// ---- PLC_MOTION/FLYING_SAW/class/FB_FlyingCtrl.TcPOU
FUNCTION_BLOCK FB_FlyingCtrl EXTENDS FB_FlyingBase IMPLEMENTS I_Fly_Ctrl
VAR
  _eInit                    : E_PROGRESS;
  _nAxisIndex               : UINT;       // know thyself
  _nMasterIndex             : UINT;       // to whom must I answer?

  // get interface from McAxis for access to Reset, Enable, Disable, Halt
  _ItfMcAxis                : ARRAY[1..PLC_CONSTANT.MAX_AXIS] OF I_McAxis;

  // pointers to all; access required for coupling; access by index
  _Ctrl                     : POINTER TO ARRAY[1..PLC_CONSTANT.MAX_AXIS] OF ST_FLY_CTRL;    // contains command to be executed
  _State                    : POINTER TO ARRAY[1..PLC_CONSTANT.MAX_AXIS] OF ST_FLY_STATE;   // mirrors command with added result

  //_Info                     : POINTER TO ARRAY[1..PLC_CONSTANT.MAX_AXIS] OF ST_FLY_INFO;    // Read Info Data
  _Data                     : POINTER TO ARRAY[1..PLC_CONSTANT.MAX_AXIS] OF ST_FLY_DATA;    // fLYINGsAW parameters

  _MoveData                 : POINTER TO ARRAY[1..PLC_CONSTANT.MAX_AXIS] OF ST_AXIS_MOVE_DATA;   // dynamic parameters

  _Options                  : POINTER TO ARRAY[1..PLC_CONSTANT.MAX_AXIS] OF ST_FLY_OPTIONS; // gear in slave options

  // local copies of command
  _eCmd,
  _eCmdOld                  : E_AXIS_CTRL;

  // execution state
  _eResult                  : E_PROGRESS;   // result of execution state
  _eResultOld               : E_PROGRESS;   // old result for detecting change
  _eState                   : E_AXIS_STATE; // execution state
END_VAR

PROPERTY AxisCtrl : pointer to ARRAY[1..PLC_CONSTANT.MAX_AXIS] OF ST_FLY_CTRL
SET
_Ctrl := AxisCtrl;
END_SET
END_PROPERTY

METHOD AxisFlyIdle : E_PROGRESS
VAR_INPUT
  Execute           : BOOL;
END_VAR
VAR_INST
  _eResult,
  _eState           : E_PROGRESS;
  _nRetry           : UINT;
END_VAR
IF NOT Execute THEN _eState := E_PROGRESS.PROGRESS_INIT; END_IF
IF NOT Check() THEN _eState := E_PROGRESS.PROGRESS_ERROR; END_IF

CASE _eState
OF
  E_PROGRESS.PROGRESS_INIT:
    IF Execute 
    THEN
      memset(ADR(_stMsg),0,SIZEOF(_stMsg));
      _nRetry                       := 0;
      _eResult                      := _ItfAxis.Reset(FALSE);
      _eState                       := E_PROGRESS.PROGRESS_BUSY;
    END_IF
END_CASE
CASE _eState
OF
  E_PROGRESS.PROGRESS_PREPARE:
    _nRetry                         := _nRetry + 1;
    _eResult                        := _ItfAxis.Reset(FALSE);
    _eResult                        := _ItfAxis.Enable(FALSE);

    _eState                         := E_PROGRESS.PROGRESS_BUSY;

    _stMsg.eType                    := E_MessageType.eMessageInfo;
    _stMsg.eSubdevice               :=  e_SubDevice.fbPower;
    _stMsg.iErrorNumber             := _nErrorId;

    _stMsg.sText                    := concat(TO_STRING(_eCmd), ' retry: ');
    _stMsg.sText                    := concat(_stMsg.sText, TO_STRING(_nRetry));

    IF (_MessageLevel < E_MessageType.eMessageError)
    THEN
      f_MessageSet(_stMsg);
    END_IF
END_CASE
CASE _eState
OF
  E_PROGRESS.PROGRESS_BUSY:
    _eResult                        := _ItfAxis.Reset(TRUE);

    IF (_eResult = E_PROGRESS.PROGRESS_DONE)
    THEN
      _eState                       := E_PROGRESS.PROGRESS_STARTUP;
    END_IF
END_CASE
CASE _eState
OF
  E_PROGRESS.PROGRESS_STARTUP:
    _eResult                        := _ItfAxis.Reset(FALSE);
    _eResult                        := _ItfAxis.Enable(FALSE);
    _eState                         := E_PROGRESS.PROGRESS_CHECK;
END_CASE
CASE _eState
OF
  E_PROGRESS.PROGRESS_CHECK:
    _eResult                        := _ItfAxis.Enable(TRUE);

    IF (_nRetry > MAX_RETRY)
    THEN
      _eState                       := E_PROGRESS.PROGRESS_ERROR;

    ELSIF (_eResult = E_PROGRESS.PROGRESS_DONE)
    THEN
      _ItfAxis.Enable(FALSE);
      _eState                       := E_PROGRESS.PROGRESS_DONE;

    ELSIF (_eResult = E_PROGRESS.PROGRESS_ERROR)
    THEN
      _eState                       := E_PROGRESS.PROGRESS_PREPARE;

      _nErrorId                     := _ItfAxis.AxisRef.NcToPlc.ErrorCode;
    
      _stMsg.eType                  := E_MessageType.eMessageError;
      _stMsg.eSubdevice             :=  e_SubDevice.fbPower;
      _stMsg.iErrorNumber           := _nErrorId;

      _stMsg.sText                  := concat(TO_STRING(_eCmd), ' error axis enable: ');
      _stMsg.sText                  := concat(_stMsg.sText, TO_STRING(_nAxisIndex));

      f_MessageSet(_stMsg);
    END_IF
END_CASE

AxisFlyIdle                         := _eState;
END_METHOD

METHOD AxisGearInPos : E_PROGRESS
VAR_INPUT
  Execute           : BOOL;
END_VAR
VAR_INST
  _eCk              : E_CHECK_STATE;

  _eResult,
  _eState           : E_PROGRESS;
  _rValue           : LREAL;
  _udiErr           : UDINT;
END_VAR
IF NOT Execute THEN _eState := E_PROGRESS.PROGRESS_INIT; END_IF
IF NOT Check() THEN _eState := E_PROGRESS.PROGRESS_ERROR; END_IF


CASE _eState
OF
  E_PROGRESS.PROGRESS_INIT:
    IF Execute 
    THEN
      _udiErr                       := 0;

      IF NOT (_nMasterIndex > 0) OR
         NOT (_nMasterIndex < PLC_CONSTANT.MAX_AXIS+1)
      THEN
        _eState                     := E_PROGRESS.PROGRESS_ERROR;
        _eCk                        := E_CHECK_STATE.FLYING_MASTER_AXIS_REF_INVALID;

        _stMsg.eType                := E_MessageType.eMessageError;
        _stMsg.eSubdevice           := e_Subdevice.FlyingSawControl;
        _stMsg.iErrorNumber         := _nMasterIndex;
  
        _stMsg.sText                := concat(' : ', TO_STRING(_eCk));
        f_MessageSet(_stMsg);

      ELSE
        _Master                     ref= _ItfMcAxis[_nMasterIndex].AxisRef;
        _eState                     := E_PROGRESS.PROGRESS_BUSY;
        _eCk                        := E_CHECK_STATE.CHECK_DONE;
        _eResult                    := GearInPos(FALSE, _stMoveData, _stFlyData, _stOptions);
      END_IF
    END_IF

  E_PROGRESS.PROGRESS_BUSY:
      _eResult                      := GearInPos(TRUE, _stMoveData, _stFlyData, _stOptions);

    IF (_eResult = E_PROGRESS.PROGRESS_ERROR) OR
       (_eResult = E_PROGRESS.PROGRESS_OCCUPIED)
    THEN
      GearInPos(FALSE, _stMoveData, _stFlyData, _stOptions);
      _eState                       := E_PROGRESS.PROGRESS_ERROR;
      _udiErr                       := _fbGearInPos.ErrorID;

    ELSIF (_eResult = E_PROGRESS.PROGRESS_DONE)
    THEN
      GearInPos(FALSE, _stMoveData, _stFlyData, _stOptions);
      _eState                       := E_PROGRESS.PROGRESS_WORKING;
    END_IF

  E_PROGRESS.PROGRESS_WORKING:
      _eState                       := E_PROGRESS.PROGRESS_DONE;
END_CASE


AxisGearInPos                       := _eState;
END_METHOD

METHOD AxisGearInVelo : E_PROGRESS
VAR_INPUT
  Execute           : BOOL;
END_VAR
VAR_INST
  _eCk              : E_CHECK_STATE;

  _eResult,
  _eState           : E_PROGRESS;
  _rValue           : LREAL;
  _udiErr           : UDINT;
END_VAR
IF NOT Execute THEN _eState := E_PROGRESS.PROGRESS_INIT; END_IF
IF NOT Check() THEN _eState := E_PROGRESS.PROGRESS_ERROR; END_IF


CASE _eState
OF
  E_PROGRESS.PROGRESS_INIT:
    IF Execute 
    THEN
      _udiErr                       := 0;

      IF NOT (_nMasterIndex > 0) OR
         NOT (_nMasterIndex < PLC_CONSTANT.MAX_AXIS+1)
      THEN
        _eState                     := E_PROGRESS.PROGRESS_ERROR;
        _eCk                        := E_CHECK_STATE.FLYING_MASTER_AXIS_REF_INVALID;

        _stMsg.eType                := E_MessageType.eMessageError;
        _stMsg.eSubdevice           := e_Subdevice.FlyingSawControl;
        _stMsg.iErrorNumber         := _nMasterIndex;
  
        _stMsg.sText                := concat(' : ', TO_STRING(_eCk));
        f_MessageSet(_stMsg);

      ELSE
        _eState                     := E_PROGRESS.PROGRESS_BUSY;
        _eCk                        := E_CHECK_STATE.CHECK_DONE;
        _eResult                    := GearInVelo(FALSE, _stMoveData, _stFlyData, _stOptions);
      END_IF
    END_IF
END_CASE
CASE _eState
OF
  E_PROGRESS.PROGRESS_BUSY:
      _eResult                      := GearInVelo(TRUE, _stMoveData, _stFlyData, _stOptions);

    IF (_eResult = E_PROGRESS.PROGRESS_ERROR)
    THEN
      GearInVelo(FALSE, _stMoveData, _stFlyData, _stOptions);
      _eState                       := E_PROGRESS.PROGRESS_ERROR;
      _udiErr                       := _fbGearInVelo.ErrorID;

    ELSIF (_eResult = E_PROGRESS.PROGRESS_DONE)
    THEN
      GearInVelo(FALSE, _stMoveData, _stFlyData, _stOptions);
      _eState                       := E_PROGRESS.PROGRESS_WORKING;
    END_IF

  E_PROGRESS.PROGRESS_WORKING:
      _eState                       := E_PROGRESS.PROGRESS_DONE;
END_CASE


AxisGearInVelo                      := _eState;
END_METHOD

PROPERTY AxisIndex : uint
SET
_nAxisIndex := AxisIndex;
END_SET
END_PROPERTY

PROPERTY AxisState : pointer to ARRAY[1..PLC_CONSTANT.MAX_AXIS] OF ST_FLY_STATE
SET
_State := AxisState;
END_SET
END_PROPERTY

METHOD PRIVATE Check : BOOL
//-----------------------------------------------------------------------------
_szSyncMode[1]            := SIZEOF(_stOptions.SyncMode);
_szSyncMode[2]            := SIZEOF(_stSyncMode);

IF NOT (_szSyncMode[1] = _szSyncMode[2])
THEN
  _eCheck                 := E_CHECK_STATE.FLYING_OPTIONS_SYNCMODE_SIZE_NOT_EQUAL;
  RETURN;
END_IF
//-----------------------------------------------------------------------------
IF (_nAxisIndex < 1) OR
   (_nAxisIndex > PLC_CONSTANT.MAX_AXIS)
THEN
  _eCheck                 := E_CHECK_STATE.AXIS_INDEX_OUT_OF_RANGE;
  RETURN;
END_IF
//-----------------------------------------------------------------------------
IF NOT (_ItfMcAxis[_nAxisIndex] <> 0)
THEN
  _eCheck                 := E_CHECK_STATE.FLYING_SLAVE_ITF_MC_AXIS_INVALID;
  RETURN;
ELSE
  _ItfAxis                := _ItfMcAxis[_nAxisIndex];
END_IF
//-----------------------------------------------------------------------------
IF NOT (_Ctrl <> 0)
THEN
  _eCheck                 := E_CHECK_STATE.AXIS_CTRL_POINTER_INVALID;
  RETURN;
END_IF
//-----------------------------------------------------------------------------
IF NOT (_State <> 0)
THEN
  _eCheck                 := E_CHECK_STATE.AXIS_STATE_POINTER_INVALID;
  RETURN;
END_IF
//-----------------------------------------------------------------------------
IF NOT (_Data <> 0)
THEN
  _eCheck                 := E_CHECK_STATE.FLYING_FLY_DATA_POINTER_INVALID;
  RETURN;
END_IF
IF NOT (_MoveData <> 0)
THEN
  _eCheck                 := E_CHECK_STATE.FLYING_MOVE_DATA_POINTER_INVALID;
  RETURN;
END_IF
IF NOT (_Options <> 0)
THEN
  _eCheck                 := E_CHECK_STATE.FLYING_OPTIONS_POINTER_INVALID;
  RETURN;
END_IF
//-----------------------------------------------------------------------------
//  NaN INF check
//-----------------------------------------------------------------------------
IF NOT IsFinite(F_LReal(_Data^[_nAxisIndex].rDelta))
THEN
  _Data^[_nAxisIndex].rDelta              := 0.0;
END_IF

IF NOT IsFinite(F_LReal(_Data^[_nAxisIndex].rDeltaToMasterPos))
THEN
  _Data^[_nAxisIndex].rDeltaToMasterPos   := 0.0;
END_IF

IF NOT IsFinite(F_LReal(_Data^[_nAxisIndex].rGearNumerator))
THEN
  _Data^[_nAxisIndex].rGearNumerator      := 0.0;
END_IF

IF NOT IsFinite(F_LReal(_Data^[_nAxisIndex].rMasterStartDistance))
THEN
  _Data^[_nAxisIndex].rMasterStartDistance := 0.0;
END_IF

IF NOT IsFinite(F_LReal(_Data^[_nAxisIndex].rModuloSyncPosSlave))
THEN
	_Data^[_nAxisIndex].rModuloSyncPosSlave  := 0.0;
END_IF
//-----------------------------------------------------------------------------
//-----------------------------------------------------------------------------
_eCheck                   := E_CHECK_STATE.CHECK_DONE;
Check                     := TRUE;
//-----------------------------------------------------------------------------
//-----------------------------------------------------------------------------
END_METHOD

//-------------------------------------------------------------------------------------
//
//  HAUD 2026 06 01
//
//  Cmd
//    - gets state for ctrl
//    - checks for eInit to be done, before any other commands are accepted
//    - prepare your commands here
//    - init what you have to here
//
//-------------------------------------------------------------------------------------
METHOD PRIVATE Cmd  : E_AXIS_STATE
VAR_INPUT
  eCmd              : E_AXIS_CTRL;
END_VAR
VAR_INST
  _IdxMaster        : UDINT;
  _stMsg            : ST_Message;
  _estate           : E_AXIS_STATE;
  _eChk             : E_CHECK_STATE;
END_VAR
_bError                               := FALSE;
CASE eCmd
OF
  //-------------------------------------------------------------------------------------
  E_AXIS_CTRL.AXIS_INIT:
    _eInit    := _eResult             := Init(FALSE);
    _estate                           := E_AXIS_STATE.AXIS_INIT;
ELSE
  IF (_eInit <> E_PROGRESS.PROGRESS_DONE)
  THEN
    _eResult                          := E_PROGRESS.PROGRESS_INVALID;
    _estate                           := E_AXIS_STATE.AXIS_NO_INIT;
  ELSE
    CASE eCmd
    OF
      //---------------------------------------------------------------------------------
      E_AXIS_CTRL.AXIS_IDLE:
        _eResult                      := AxisFlyIdle(FALSE);
        _estate                       := E_AXIS_STATE.AXIS_IDLE;

      //---------------------------------------------------------------------------------
      E_AXIS_CTRL.FLY_GEAR_IN_POS:
        _IdxMaster                    := GetIndex(_Data^[_nAxisIndex].nMasterAxisId);
        _nMasterIndex                 := TO_UINT(_IdxMaster);
        _stFlyData                    := _Data^[_nAxisIndex];
        _stMoveData                   := _MoveData^[_nAxisIndex];
        _stOptions                    := _Options^[_nAxisIndex];

        IF (_IdxMaster = 0)
        THEN
          _eResult                    := E_PROGRESS.PROGRESS_ERROR;
          _eChk                       := E_CHECK_STATE.FLYING_MASTER_AXIS_REF_INVALID;
  
          _stMsg.eType                := E_MessageType.eMessageError;
          _stMsg.eSubdevice           := e_Subdevice.FlyingSawControl;
          _stMsg.iErrorNumber         := _nMasterIndex;
    
          _stMsg.sText                := concat(' : ', TO_STRING(_eChk));
          f_MessageSet(_stMsg);
        ELSE
          _eChk                       := _eCheck;
          _eResult                    := AxisGearInPos(FALSE);
          _estate                     := E_AXIS_STATE.FLY_GEAR_IN_POS;
        END_IF

      //---------------------------------------------------------------------------------
      E_AXIS_CTRL.FLY_GEAR_IN_VELO:
        _IdxMaster                    := GetIndex(_Data^[_nAxisIndex].nMasterAxisId);
        _stFlyData                    := _Data^[_nAxisIndex];
        _stMoveData                   := _MoveData^[_nAxisIndex];
        _stOptions                    := _Options^[_nAxisIndex];

        IF (_IdxMaster = 0)
        THEN
          _eResult                    := E_PROGRESS.PROGRESS_ERROR;
          _eChk                       := E_CHECK_STATE.FLYING_MASTER_AXIS_REF_INVALID;
  
          _stMsg.eType                := E_MessageType.eMessageError;
          _stMsg.eSubdevice           := e_Subdevice.FlyingSawControl;
          _stMsg.iErrorNumber         := _nMasterIndex;
    
          _stMsg.sText                := concat(' : ', TO_STRING(_eChk));
          f_MessageSet(_stMsg);
        ELSE
          _eChk                       := _eCheck;
          _eResult                    := AxisGearInVelo(FALSE);
          _estate                     := E_AXIS_STATE.FLY_GEAR_IN_VELO;
        END_IF

    //-----------------------------------------------------------------------------------
    ELSE
      _estate                         := E_AXIS_STATE.AXIS_NULL;

      IF (eCmd = E_AXIS_CTRL.AXIS_NULL)
      THEN
        _eResult                      := E_PROGRESS.PROGRESS_DONE;
      ELSE
        _eResult                      := E_PROGRESS.PROGRESS_INVALID;
  
        _stMsg.eType                  := E_MessageType.eMessageError;
        _stMsg.eSubdevice             := e_Subdevice.FlyingSawControl;
        _stMsg.iErrorNumber           := 0;
  
        _stMsg.sText                  := 'E_AXIS_CTRL.';
        _stMsg.sText                  := concat(_stMsg.sText, TO_STRING(eCmd));
        _stMsg.sText                  := concat(_stMsg.sText, ': ');
        _stMsg.sText                  := concat(_stMsg.sText, TO_STRING(_eResult));

        f_MessageSet(_stMsg);
      END_IF
    END_CASE
  END_IF // _eInit
END_CASE

Cmd                                   := _estate;
END_METHOD

METHOD Cycle  : e_progress
VAR_INST
  _eCycle     : E_PROGRESS;

  _eCheckOld  : E_CHECK_STATE;
END_VAR
IF NOT Check() THEN Cycle := _eCycle := _eResult := E_PROGRESS.PROGRESS_ERROR; END_IF
//-----------------------------------------------------------------------------
//  set message device
//-----------------------------------------------------------------------------
_stMsg.eDevice                      := e_Device.FlyingSaw + (_ItfAxis.AxisRef.NcToPlc.AxisId);
//-----------------------------------------------------------------------------
//-----------------------------------------------------------------------------
// OnChange log _eCheck; in case of error --> return to caller
//-----------------------------------------------------------------------------
IF (_eCheck <> _eCheckOld)
THEN
  LogCheck();
  _eCheckOld                        := _eCheck;
END_IF
//-----------------------------------------------------------------------------
IF NOT (_eCheck = E_CHECK_STATE.CHECK_DONE)
THEN
  RETURN;
END_IF
//-----------------------------------------------------------------------------
//-----------------------------------------------------------------------------
// get command from outside world
//-----------------------------------------------------------------------------
_eCmd                               := _Ctrl^[_nAxisIndex].eCmd;
//-----------------------------------------------------------------------------
//-----------------------------------------------------------------------------
//  OnChange react to command
//-----------------------------------------------------------------------------
IF (_eCmd <> _eCmdOld)
THEN
  // get busy
  _eState                           := Cmd(_eCmd); // get execution state for command
  _eCmdOld                          := _eCmd;
  LogControl();
END_IF
//-----------------------------------------------------------------------------
//-----------------------------------------------------------------------------
//  execution result
//-----------------------------------------------------------------------------
CASE _eResult
OF
  E_PROGRESS.PROGRESS_INVALID:
    _State^[_nAxisIndex].eState     := TO_UINT(E_PROGRESS.PROGRESS_ERROR);

  E_PROGRESS.PROGRESS_ERROR:
    _State^[_nAxisIndex].eState     := _eState + E_PROGRESS.PROGRESS_ERROR;

  E_PROGRESS.PROGRESS_DONE:
    _State^[_nAxisIndex].eState     := _eState + E_PROGRESS.PROGRESS_DONE;

ELSE
    _State^[_nAxisIndex].eState     := _eState + _eResult;
  //-----------------------------------------------------------------------------
  //-----------------------------------------------------------------------------
  //  execution state for command
  //-----------------------------------------------------------------------------
  CASE _eState
  OF
    //---------------------------------------------------------------------------
    E_AXIS_STATE.AXIS_INIT:
      // axis always requires one init from outside world at startup
      // _eInit has to be valid for other commands to be accepted in Cmd(_eCtrl)
      _eInit := _eResult            := Init(TRUE);
  
    //---------------------------------------------------------------------------
    E_AXIS_STATE.AXIS_NO_INIT:
      // we are here because you sent a command before having done INIT
      _eResult                      := E_PROGRESS.PROGRESS_ERROR;
  
    //---------------------------------------------------------------------------
    E_AXIS_STATE.AXIS_IDLE:
      _eResult                      := AxisFlyIdle(TRUE);
  
    //---------------------------------------------------------------------------
    E_AXIS_STATE.FLY_GEAR_IN_POS:
      _eResult                      := AxisGearInPos(TRUE);
  
    //---------------------------------------------------------------------------
    E_AXIS_STATE.FLY_GEAR_IN_VELO:
      _eResult                      := AxisGearInVelo(TRUE);

  ELSE
    IF (_eCmd > E_AXIS_CTRL.AXIS_NULL)
    THEN
      _eResult                      := E_PROGRESS.PROGRESS_NOT_EXIST;
    ELSE
      _eResult                      := E_PROGRESS.PROGRESS_INVALID;
    END_IF
  END_CASE
END_CASE
//-----------------------------------------------------------------------------
//-----------------------------------------------------------------------------
//  OnChange of execution state result
//    - log result and clear error number on interface
//-----------------------------------------------------------------------------
IF (_eResult <> _eResultOld)
THEN
  LogResult();
  _eResultOld                       := _eResult;
END_IF
//-----------------------------------------------------------------------------
END_METHOD

PROPERTY GearData : pointer to ARRAY[1..PLC_CONSTANT.MAX_AXIS] OF ST_FLY_DATA
SET
_Data := GearData;
END_SET
END_PROPERTY

METHOD GetIndex : udint
VAR_INPUT
  AxisId        : UDINT;
END_VAR
VAR
  _nidx         : UDINT;
END_VAR
IF NOT Check() THEN GetIndex := 0; RETURN; END_IF

FOR _nidx := 1 TO PLC_CONSTANT.MAX_AXIS
DO
  IF (_ItfMcAxis[_nidx].AxisRef.NcToPlc.AxisId = AxisId)
  THEN
    GetIndex      := _nIdx;
    RETURN;
  END_IF
END_FOR

GetIndex          := 0;
END_METHOD

METHOD PRIVATE Init : E_PROGRESS
VAR_INPUT
  Execute           : BOOL;
END_VAR
VAR_INST
  _eResult,
  _eState           : E_PROGRESS;
  _rValue           : LREAL;
END_VAR
IF NOT Execute THEN Init := _estate := E_PROGRESS.PROGRESS_INIT; END_IF
IF NOT Check() THEN Init := _estate := E_PROGRESS.PROGRESS_ERROR; END_IF

CASE _eState
OF
  E_PROGRESS.PROGRESS_INIT:
    IF Execute 
    THEN
      memset(ADR(_stMsg),0,SIZEOF(_stMsg));

      _nErrorId                     := 0;
      _rValue                       := 0;
      _eState                       := E_PROGRESS.PROGRESS_BUSY;
    END_IF
END_CASE
CASE _eState
OF
  E_PROGRESS.PROGRESS_BUSY:
    _eState                         := E_PROGRESS.PROGRESS_STARTUP;
END_CASE
CASE _eState
OF
  E_PROGRESS.PROGRESS_STARTUP:
    // keep this for future use
    _eResult                        := E_PROGRESS.PROGRESS_DONE;//StartUp(TRUE);
    IF (_eResult = E_PROGRESS.PROGRESS_DONE)
    THEN
      _eState                       := E_PROGRESS.PROGRESS_PREPARE;
      _ItfMcAxis[_nAxisIndex].Reset(FALSE);
    ELSIF (_eResult = E_PROGRESS.PROGRESS_ERROR)
    THEN
      _eState                       := _eResult;

      _stMsg.eType                  := E_MessageType.eMessageError;
      _stMsg.eDevice                := e_Device.FlyingSaw + (_ItfAxis.AxisRef.NcToPlc.AxisId);
      _stMsg.eSubdevice             := e_Subdevice.FlyingSawStartUp;
      _stMsg.iErrorNumber := _nErrorId  := 6666;

      _stMsg.sText                  := TO_STRING(_eState);
      f_MessageSet(_stMsg);
    END_IF
END_CASE
CASE _eState
OF
  E_PROGRESS.PROGRESS_PREPARE:
    _eResult                        := _ItfMcAxis[_nAxisIndex].Reset(TRUE);
    IF (_eResult = E_PROGRESS.PROGRESS_DONE)
    THEN
      _eState                       := E_PROGRESS.PROGRESS_CHECK;
    ELSIF (_eResult = E_PROGRESS.PROGRESS_ERROR)
    THEN
      _eState                       := _eResult;

      _stMsg.eType                  := E_MessageType.eMessageError;
      _stMsg.eDevice                := e_Device.FlyingSaw + (_ItfAxis.AxisRef.NcToPlc.AxisId);
      _stMsg.eSubdevice             := e_Subdevice.fbReset;
      _stMsg.iErrorNumber           := _ItfAxis.AxisRef.Status.ErrorID;

      _stMsg.sText                  := TO_STRING(_eState);
      f_MessageSet(_stMsg);
    END_IF
END_CASE
CASE _eState
OF
  E_PROGRESS.PROGRESS_CHECK:
    _eResult                        := _ItfMcAxis[_nAxisIndex].Reset(FALSE);
    _eState                         := E_PROGRESS.PROGRESS_OCCUPIED;
END_CASE
CASE _eState
OF
  E_PROGRESS.PROGRESS_OCCUPIED:
    _eState                         := E_PROGRESS.PROGRESS_WORKING;
END_CASE
CASE _eState
OF
  E_PROGRESS.PROGRESS_WORKING:
    _eState                         := E_PROGRESS.PROGRESS_DONE;

    _stMsg.eType                    := E_MessageType.eMessageInfo;
    _stMsg.eSubdevice               := e_Subdevice.FlyingSawControl;
    _stMsg.iErrorNumber             := 0;
    _stMsg.sText                    := concat('Init: ', TO_STRING(_eState));

    IF (_MessageLevel < E_MessageType.eMessageError)
    THEN
      f_MessageSet(_stMsg);
    END_IF
END_CASE

Init                                := _eState;
END_METHOD

PROPERTY ItfMcAxes : array[1..MAX_AXIS] of I_McAxis
SET
_ItfMcAxis := ItfMcAxes;
END_SET
END_PROPERTY

METHOD LogCheck
VAR_INST
  _sChck            : STRING(40);
END_VAR
  _stMsg.eType               := SEL((_eCheck = E_CHECK_STATE.CHECK_DONE),(E_MessageType.eMessageError),(E_MessageType.eMessageInfo));
  _stMsg.eSubdevice          := e_Subdevice.FlyingSawControl;
  _stMsg.iErrorNumber        := _nAxisIndex;

  _sChck                     := concat('E_CHECK_STATE', '.');
  _sChck                     := concat(_sChck, TO_STRING(_eCheck));

  _stMsg.sText               := concat('cyclic check: ', _sChck);

  IF (_MessageLevel > E_MessageType.eMessageError)
  THEN
    f_MessageSet(_stMsg);
  ELSE
    IF (_stMsg.eType = E_MessageType.eMessageError)
    THEN
      f_MessageSet(_stMsg);
    END_IF
  END_IF
END_METHOD

METHOD PRIVATE LogControl
VAR_INST
  _sResult,
  _sCtrl            : STRING(40);
END_VAR
  _stMsg.eType               := E_MessageType.eMessageInfo;
  _stMsg.eDevice             := E_Device.FlyingSaw + (_ItfAxis.AxisRef.NcToPlc.AxisId);
  _stMsg.eSubdevice          := e_Subdevice.FlyingSawControl;
  _stMsg.iErrorNumber        := _nAxisIndex;

  _sCtrl                     := concat('E_AXIS_CTRL', '.');
  _sCtrl                     := concat(_sCtrl, TO_STRING(_eCmd));

  _stMsg.sText               := concat('new command: ', _sCtrl);

  IF (_MessageLevel > E_MessageType.eMessageError)
  THEN
    f_MessageSet(_stMsg);
  ELSE
    IF (_stMsg.eType = E_MessageType.eMessageError)
    THEN
      f_MessageSet(_stMsg);
    END_IF
  END_IF
END_METHOD

METHOD PRIVATE LogResult
VAR_INST
  _sResult,
  _sCtrl            : STRING(40);
END_VAR
  _stMsg.eType               := E_MessageType.eMessageInfo;
  _stMsg.eDevice             := E_Device.FlyingSaw + (_ItfAxis.AxisRef.NcToPlc.AxisId);
  _stMsg.eSubdevice          := e_Subdevice.FlyingSawControl;
  _stMsg.iErrorNumber        := _nAxisIndex;

  _sCtrl                     := concat('E_AXIS_CTRL', '.');
  _sCtrl                     := concat(_sCtrl, TO_STRING(_eCmdOld));

  _sResult                   := concat(': E_PROGRESS', '.');
  _sResult                   := concat(_sResult, TO_STRING(_eResult));

  _stMsg.sText               := concat(_sCtrl, ' ');
  _stMsg.sText               := concat(_sCtrl, _sResult);

  IF (_MessageLevel > E_MessageType.eMessageError)
  THEN
    f_MessageSet(_stMsg);
  ELSE
    IF (_stMsg.eType = E_MessageType.eMessageError)
    THEN
      f_MessageSet(_stMsg);
    END_IF
  END_IF
END_METHOD

PROPERTY MoveData : pointer to ARRAY[1..PLC_CONSTANT.MAX_AXIS] OF ST_AXIS_MOVE_DATA
SET
_MoveData := MoveData;
END_SET
END_PROPERTY

PROPERTY Options : pointer to ARRAY[1..PLC_CONSTANT.MAX_AXIS] OF ST_FLY_OPTIONS
SET
_Options := Options;
END_SET
END_PROPERTY

END_FUNCTION_BLOCK

// ---- PLC_MOTION/FUNCTIONS/TOUCH_PROBE/FB_TouchProbe.TcPOU
FUNCTION_BLOCK FB_TouchProbe EXTENDS FB_Xfc
VAR
  _Ctrl             : REFERENCE TO ARRAY[1..MAX_TOUCH_PROBE] OF ST_CTRL_TOUCH_PROBE;
  _State            : REFERENCE TO ARRAY[1..MAX_TOUCH_PROBE] OF ST_STATE_TOUCH_PROBE;

  _Input            : POINTER TO ARRAY[1..MAX_TOUCH_PROBE] OF ST_MTI_Input;
  _InputState       : POINTER TO ARRAY[1..MAX_TOUCH_PROBE] OF ST_MTI_STATUS;

  _Index            : UDINT;
  _AxisId           : UDINT;
  _AxisIndex        : UDINT;

  _CtrlLocal        : ST_CTRL_TOUCH_PROBE;  // control data is copied to local on start of function
  _McDirection      : Tc2_MC2.MC_Direction;

  _eStateProgress   : E_PROGRESS;
  _eResult          : E_PROGRESS;

  _rtrigEnable      : Tc2_Standard.R_TRIG;
  _TrigCount        : UDINT;

  _CurrentTime      : ULINT;
  _CurrentTimeShort : UDINT;
  _LatchTime        : UDINT;
  _LatchState       : Bool;

  _bError           : BOOL;
  _stMsg            : ST_Message;
  _MessageLevel     : E_MessageType;
END_VAR

PROPERTY Ctrl : REFERENCE TO ARRAY [1..MAX_TOUCH_PROBE] OF ST_CTRL_TOUCH_PROBE
SET
_Ctrl REF= Ctrl;
END_SET
END_PROPERTY

METHOD Cycle : BOOL
VAR_INPUT
END_VAR
//-----------------------------------------------------------------------------
//-----------------------------------------------------------------------------
//  Check Enable
//-----------------------------------------------------------------------------
IF NOT _Ctrl[_Index].Enable
THEN
  // clear function state if not enabled
  _eStateProgress                   := E_PROGRESS.PROGRESS_INVALID;
  _LatchState                       := FALSE;
  _State[_Index].State              := TO_UINT(_eStateProgress);
END_IF
//-----------------------------------------------------------------------------
//-----------------------------------------------------------------------------
//  set message device
//-----------------------------------------------------------------------------
_eDeviceFunction                    := e_Device.XfcTouchProbe + _Index;
//-----------------------------------------------------------------------------
//-----------------------------------------------------------------------------
//  rising trigger react to enable command
//-----------------------------------------------------------------------------
_rtrigEnable(CLK                    := _Ctrl[_Index].Enable);
//-----------------------------------------------------------------------------
//-----------------------------------------------------------------------------
//  main state machine
//-----------------------------------------------------------------------------
CASE _eStateProgress
OF
  E_PROGRESS.PROGRESS_INVALID:      // check input data
    IF _rtrigEnable.Q
    THEN
      _State[_Index].State          := TO_UINT(E_PROGRESS.PROGRESS_BUSY);
      _State[_Index].LatchPositive  := 0.0;
      _State[_Index].LatchNegative  := 0.0;

      _bError                       := FALSE;
      _eStateProgress               := E_PROGRESS.PROGRESS_INIT;

      _CtrlLocal                    := _Ctrl[_Index];   // copy control data to local, you may write new data onto struct as long as .Enable stays TRUE
      _CurrentTime                  := Tc2_EtherCAT.F_GetCurDcTickTime64();
      _CurrentTimeShort             := TO_UDINT(_CurrentTime AND 16#FFFFFFFF);

      _AxisId                       := _CtrlLocal.AxisId;   // TwinCAT NC AxisId
      _AxisIndex                    := GetIndex(_AxisId);   // corresponding index in axis array

      _stMsg.iErrorNumber           := 0;

      IF NOT (_AxisIndex > 0) OR NOT (_AxisId > 0)
      THEN
        _bError                     := TRUE;
        _stMsg.iErrorNumber         := 1;
        _stMsg.sText                := 'AxisId Invalid ';
        _eStateProgress             := E_PROGRESS.PROGRESS_STILL_WORKING;
      END_IF

      IF NOT (_CtrlLocal.Direction = MC_Positive_Direction) OR 
         NOT (_CtrlLocal.Direction = MC_Negative_Direction)
      THEN
        _bError                     := TRUE;
        _stMsg.iErrorNumber         := 2;
        _stMsg.sText                := 'Direction Invalid ';
        _eStateProgress             := E_PROGRESS.PROGRESS_STILL_WORKING;
      END_IF

      IF NOT IsFinite(F_LReal(_CtrlLocal.PositionStart))
      THEN
        _bError                     := TRUE;
        _stMsg.iErrorNumber         := 3;
        _stMsg.sText                := 'PositionStart not finite ';
        _eStateProgress             := E_PROGRESS.PROGRESS_STILL_WORKING;
      END_IF

      IF NOT IsFinite(F_LReal(_CtrlLocal.PositionEnd))
      THEN
        _bError                     := TRUE;
        _stMsg.iErrorNumber         := 4;
        _stMsg.sText                := 'PositionEnd not finite ';
        _eStateProgress             := E_PROGRESS.PROGRESS_STILL_WORKING;
      END_IF
    END_IF

  E_PROGRESS.PROGRESS_INIT:
      _eDeviceAxis                  := e_Device.XfcAxis + (_CtrlLocal.AxisId);
      _eStateProgress               := E_PROGRESS.PROGRESS_BUSY;

      IF (_MessageLevel = E_MessageType.eMessageVerbose)
      THEN
        _stMsg.eType                := E_MessageType.eMessageVerbose;
        _stMsg.eDevice              := _eDeviceFunction;
        _stMsg.eSubdevice           := e_Subdevice.XfcTouchProbe;
        _stMsg.iErrorNumber         := _eDeviceAxis;
        _stMsg.sText                := concat(TO_STRING(_eStateProgress), ': ');
        _stMsg.sText                := concat(_stMsg.sText, TO_STRING(e_Device.XfcAxis));
        _stMsg.sText                := concat(_stMsg.sText, '_ID_');
        _stMsg.sText                := concat(_stMsg.sText, TO_STRING(_AxisId));

        f_MessageSet(_stMsg);
      END_IF
END_CASE
//-----------------------------------------------------------------------------
//-----------------------------------------------------------------------------
CASE _eStateProgress
OF
  E_PROGRESS.PROGRESS_BUSY:
    _McDirection                    := _CtrlLocal.Direction;
    CASE _McDirection
    OF
      MC_Positive_Direction:
        IF (_ItfAxis[_AxisIndex].Position >= _CtrlLocal.PositionStart)
        THEN
          _eResult                  := PositionAtTime(FALSE, _CtrlLocal.AxisId, 0, _MessageLevel);
          _eStateProgress           := E_PROGRESS.PROGRESS_PREPARE;
        END_IF

      MC_Negative_Direction:
        IF (_ItfAxis[_AxisIndex].Position <= _CtrlLocal.PositionStart)
        THEN
          _eResult                  := PositionAtTime(FALSE, _CtrlLocal.AxisId, 0, _MessageLevel);
          _eStateProgress           := E_PROGRESS.PROGRESS_PREPARE;
        END_IF
    END_CASE
END_CASE
//-----------------------------------------------------------------------------
//-----------------------------------------------------------------------------
CASE _eStateProgress
OF
  E_PROGRESS.PROGRESS_PREPARE:
    CASE _McDirection
    OF
      MC_Positive_Direction:
        IF (_ItfAxis[_AxisIndex].Position > _CtrlLocal.PositionEnd)
        THEN
          _bError                   := TRUE;
          _stMsg.iErrorNumber       := 5;
          _stMsg.sText              := 'PositionEnd reached, no rising trigger ';
          _eStateProgress           := E_PROGRESS.PROGRESS_STILL_WORKING;
    
        ELSIF (_Input^[_Index].EventState) OR
              (_Input^[_Index].EventTime > _CurrentTimeShort)
        THEN
          _LatchState               := _Input^[_Index].EventState;
          _LatchTime                := _Input^[_Index].EventTime;
    
          IF (_MessageLevel = E_MessageType.eMessageVerbose)
          THEN
            _stMsg.eType            := E_MessageType.eMessageVerbose;
            _stMsg.eDevice          := _eDeviceFunction;
            _stMsg.eSubdevice       := e_Subdevice.XfcTouchProbe;
            _stMsg.iErrorNumber     := _LatchTime;
            _stMsg.sText            := concat(TO_STRING(_eStateProgress), ': ');
            _stMsg.sText            := concat(_stMsg.sText, TO_STRING(e_Device.XfcAxis));
    
            f_MessageSet(_stMsg);
          END_IF
          _eStateProgress           := E_PROGRESS.PROGRESS_STARTUP;
        END_IF

      MC_Negative_Direction:
        IF (_ItfAxis[_AxisIndex].Position < _CtrlLocal.PositionEnd)
        THEN
          _bError                   := TRUE;
          _stMsg.iErrorNumber       := 5;
          _stMsg.sText              := 'PositionEnd reached, no rising trigger ';
          _eStateProgress           := E_PROGRESS.PROGRESS_STILL_WORKING;
    
        ELSIF (_Input^[_Index].EventState) OR
              (_Input^[_Index].EventTime > _CurrentTimeShort)
        THEN
          _LatchState               := _Input^[_Index].EventState;
          _LatchTime                := _Input^[_Index].EventTime;
    
          IF (_MessageLevel = E_MessageType.eMessageVerbose)
          THEN
            _stMsg.eType            := E_MessageType.eMessageVerbose;
            _stMsg.eDevice          := _eDeviceFunction;
            _stMsg.eSubdevice       := e_Subdevice.XfcTouchProbe;
            _stMsg.iErrorNumber     := _LatchTime;
            _stMsg.sText            := concat(TO_STRING(_eStateProgress), ': ');
            _stMsg.sText            := concat(_stMsg.sText, TO_STRING(e_Device.XfcAxis));
    
            f_MessageSet(_stMsg);
          END_IF
          _eStateProgress           := E_PROGRESS.PROGRESS_STARTUP;
        END_IF
    END_CASE
END_CASE
//-----------------------------------------------------------------------------
//-----------------------------------------------------------------------------
CASE _eStateProgress
OF
  E_PROGRESS.PROGRESS_STARTUP:
    _eResult                        := PositionAtTime(TRUE, _CtrlLocal.AxisId, _LatchTime, _MessageLevel);

    IF (_eResult = E_PROGRESS.PROGRESS_ERROR)
    THEN
      _bError                       := TRUE;
      _stMsg.iErrorNumber           := 7;
      _stMsg.sText                  := 'PositionAtTime LatchPositive ';
      _eStateProgress               := E_PROGRESS.PROGRESS_STILL_WORKING;
      _eResult                      := PositionAtTime(FALSE, _CtrlLocal.AxisId, 0, _MessageLevel);

    ELSIF (_eResult = E_PROGRESS.PROGRESS_DONE)
    THEN
      _State[_Index].LatchPositive  := _XfcRecordedPosition[_AxisIndex];

      _CurrentTime                  := Tc2_EtherCAT.F_GetCurDcTickTime64();
      _CurrentTimeShort             := TO_UDINT(_CurrentTime AND 16#FFFFFFFF);

      IF (_MessageLevel = E_MessageType.eMessageVerbose)
      THEN
        _stMsg.eType                := E_MessageType.eMessageVerbose;
        _stMsg.eDevice              := _eDeviceFunction;
        _stMsg.eSubdevice           := e_Subdevice.XfcTouchProbe;
        _stMsg.iErrorNumber         := _LatchTime;
        _stMsg.sText                := concat(TO_STRING(_eStateProgress), ': ');
        _stMsg.sText                := concat(_stMsg.sText, TO_STRING(_XfcRecordedPosition[_AxisIndex]));

        f_MessageSet(_stMsg);
      END_IF
      _eStateProgress               := E_PROGRESS.PROGRESS_CHECK;
      _eResult                      := PositionAtTime(FALSE, _CtrlLocal.AxisId, 0, _MessageLevel);
    END_IF
END_CASE
//-----------------------------------------------------------------------------
//-----------------------------------------------------------------------------
CASE _eStateProgress
OF
  E_PROGRESS.PROGRESS_CHECK:
    CASE _McDirection
    OF
      MC_Positive_Direction:
        IF (_ItfAxis[_AxisIndex].Position > _CtrlLocal.PositionEnd)
        THEN
          _bError                   := TRUE;
          _stMsg.iErrorNumber       := 6;
          _stMsg.sText              := concat('PositionEnd reached, no falling trigger :', TO_STRING(_ItfAxis[_AxisIndex].Position));
          _eStateProgress           := E_PROGRESS.PROGRESS_STILL_WORKING;
    
        ELSIF NOT (_Input^[_Index].EventState) OR
              (_Input^[_Index].EventTime > _LatchTime - 1_000)
        THEN
          _LatchState               := _Input^[_Index].EventState;
          _LatchTime                := _Input^[_Index].EventTime;
    
          IF (_MessageLevel = E_MessageType.eMessageVerbose)
          THEN
            _stMsg.eType            := E_MessageType.eMessageVerbose;
            _stMsg.eDevice          := _eDeviceFunction;
            _stMsg.eSubdevice       := e_Subdevice.XfcTouchProbe;
            _stMsg.iErrorNumber     := _LatchTime;
            _stMsg.sText            := concat(TO_STRING(_eStateProgress), ': ');
            _stMsg.sText            := concat(_stMsg.sText, TO_STRING(e_Device.XfcAxis));
    
            f_MessageSet(_stMsg);
          END_IF
          _eStateProgress           := E_PROGRESS.PROGRESS_OCCUPIED;
        END_IF

      MC_Negative_Direction:
        IF (_ItfAxis[_AxisIndex].Position < _CtrlLocal.PositionEnd)
        THEN
          _bError                   := TRUE;
          _stMsg.iErrorNumber       := 6;
          _stMsg.sText              := concat('PositionEnd reached, no falling trigger :', TO_STRING(_ItfAxis[_AxisIndex].Position));
          _eStateProgress           := E_PROGRESS.PROGRESS_STILL_WORKING;
    
        ELSIF NOT (_Input^[_Index].EventState) OR
              (_Input^[_Index].EventTime > _LatchTime - 1_000)
        THEN
          _LatchState               := _Input^[_Index].EventState;
          _LatchTime                := _Input^[_Index].EventTime;
    
          IF (_MessageLevel = E_MessageType.eMessageVerbose)
          THEN
            _stMsg.eType            := E_MessageType.eMessageVerbose;
            _stMsg.eDevice          := _eDeviceFunction;
            _stMsg.eSubdevice       := e_Subdevice.XfcTouchProbe;
            _stMsg.iErrorNumber     := _LatchTime;
            _stMsg.sText            := concat(TO_STRING(_eStateProgress), ': ');
            _stMsg.sText            := concat(_stMsg.sText, TO_STRING(e_Device.XfcAxis));
    
            f_MessageSet(_stMsg);
          END_IF
          _eStateProgress           := E_PROGRESS.PROGRESS_OCCUPIED;
        END_IF
    END_CASE
END_CASE
//-----------------------------------------------------------------------------
//-----------------------------------------------------------------------------
CASE _eStateProgress
OF
  E_PROGRESS.PROGRESS_OCCUPIED:
    _eResult                        := PositionAtTime(TRUE, _CtrlLocal.AxisId, _LatchTime, _MessageLevel);

    IF (_eResult = E_PROGRESS.PROGRESS_ERROR)
    THEN
      _bError                       := TRUE;
      _stMsg.iErrorNumber           := 8;
      _stMsg.sText                  := 'PositionAtTime LatchNegative: ';
      _eStateProgress               := E_PROGRESS.PROGRESS_STILL_WORKING;
      _eResult                      := PositionAtTime(FALSE, _CtrlLocal.AxisId, 0, _MessageLevel);

    ELSIF (_eResult = E_PROGRESS.PROGRESS_DONE)
    THEN
      _State[_Index].LatchNegative  := _XfcRecordedPosition[_AxisIndex];

      IF (_MessageLevel = E_MessageType.eMessageVerbose)
      THEN
        _stMsg.eType                := E_MessageType.eMessageVerbose;
        _stMsg.eDevice              := _eDeviceFunction;
        _stMsg.eSubdevice           := e_Subdevice.XfcTouchProbe;
        _stMsg.iErrorNumber         := _LatchTime;
        _stMsg.sText                := concat(TO_STRING(_eStateProgress), ': ');
        _stMsg.sText                := concat(_stMsg.sText, TO_STRING(_XfcRecordedPosition[_AxisIndex]));

        f_MessageSet(_stMsg);
      END_IF
      _eStateProgress               := E_PROGRESS.PROGRESS_WORKING;
      _eResult                      := PositionAtTime(FALSE, _CtrlLocal.AxisId, 0, _MessageLevel);
    END_IF
END_CASE
//-----------------------------------------------------------------------------
//-----------------------------------------------------------------------------
CASE _eStateProgress
OF
  E_PROGRESS.PROGRESS_WORKING:
    _eStateProgress                 := E_PROGRESS.PROGRESS_STILL_WORKING;
END_CASE
//-----------------------------------------------------------------------------
//-----------------------------------------------------------------------------
CASE _eStateProgress
OF
  E_PROGRESS.PROGRESS_STILL_WORKING:
    IF NOT _bError
    THEN
      _eStateProgress               := E_PROGRESS.PROGRESS_DONE;

      IF (_MessageLevel > E_MessageType.eMessageWarning)
      THEN
        _stMsg.eType                := E_MessageType.eMessageInfo;
        _stMsg.eDevice              := _eDeviceFunction;
        _stMsg.eSubdevice           := e_Subdevice.XfcTouchProbe;
        _stMsg.iErrorNumber         := _eDeviceAxis;
        _stMsg.sText                := concat(TO_STRING(_eStateProgress), ': ');
        _stMsg.sText                := concat(_stMsg.sText, TO_STRING(e_Device.XfcAxis));
        _stMsg.sText                := concat(_stMsg.sText, '_ID_');
        _stMsg.sText                := concat(_stMsg.sText, TO_STRING(_AxisId));

        f_MessageSet(_stMsg);
      END_IF
      _State[_Index].State          := TO_UINT(_eStateProgress);
    ELSE
      _eStateProgress               := E_PROGRESS.PROGRESS_ERROR;

      _stMsg.eType                  := E_MessageType.eMessageError;
      _stMsg.eDevice                := _eDeviceFunction;
      _stMsg.eSubdevice             := e_Subdevice.XfcTouchProbe;
      _stMsg.sText                  := concat(_stMsg.sText, TO_STRING(_eStateProgress));
      _stMsg.sText                  := concat(_stMsg.sText, ': ');
      _stMsg.sText                  := concat(_stMsg.sText, TO_STRING(e_Device.XfcAxis));
      _stMsg.sText                  := concat(_stMsg.sText, '_ID_');
      _stMsg.sText                  := concat(_stMsg.sText, TO_STRING(_AxisId));

      f_MessageSet(_stMsg);
      _State[_Index].State          := TO_UINT(_eStateProgress) + TO_UINT(_stMsg.iErrorNumber);
    END_IF
END_CASE
END_METHOD

PROPERTY Index : udint
GET
Index := _Index;
END_GET
SET
_Index := Index;
END_SET
END_PROPERTY

PROPERTY Input : pointer TO ARRAY [1..MAX_TOUCH_PROBE] OF ST_MTI_Input
SET
_Input := Input;
END_SET
END_PROPERTY

PROPERTY InputState : pointer TO ARRAY [1..MAX_TOUCH_PROBE] OF ST_MTI_STATUS
SET
_InputState := InputState;
END_SET
END_PROPERTY

PROPERTY MessageLevel : e_messagetype
GET
MessageLevel := _MessageLevel;
END_GET
SET
_MessageLevel := MessageLevel;
END_SET
END_PROPERTY

PROPERTY State :  REFERENCE TO ARRAY[1..MAX_TOUCH_PROBE] OF ST_STATE_TOUCH_PROBE;
SET
_State REF= State;
END_SET
END_PROPERTY

END_FUNCTION_BLOCK

// ---- PLC_MOTION/XFC/FB_Xfc.TcPOU
//-----------------------------------------------------------------------------------------------------------
// XFC base class
//
// HAUD
// 18.07.2024
// - encapsulation of XFC library: Tc2_MC2_XFC
//-----------------------------------------------------------------------------------------------------------
FUNCTION_BLOCK abstract FB_Xfc
VAR
  _eDeviceFunction            : e_Device;
  _eDeviceAxis                : e_Device;

  _XfcTaskTime_DC             : T_DCTIME;

  _ItfAxis                    : ARRAY[1..MAX_AXIS] OF I_McAxis;

  // base function blocks per axis
  _XfcPositionAtTime          : ARRAY[1..MAX_AXIS] OF Tc2_MC2_XFC.XFC_PositionAtTime;
  _XfcTimeOfPosition          : ARRAY[1..MAX_AXIS] OF Tc2_MC2_XFC.XFC_TimeOfPosition;
  _XfcTimeToPosition          : ARRAY[1..MAX_AXIS] OF Tc2_MC2_XFC.XFC_TimeToPosition;
  _XfcTimeToModuloPosition    : ARRAY[1..MAX_AXIS] OF Tc2_MC2_XFC.XFC_TimeToModuloPosition;

  _XfcNcTimeConversionOptions : ARRAY[1..MAX_AXIS] OF ST_NcTimeConversionOptions; 
  _XfcRecordedPosition        : ARRAY[1..MAX_AXIS] OF LREAL;
  _XfcRecordedTime            : ARRAY[1..MAX_AXIS] OF T_DCTIME32;

  _XfcDurationToPosition      : ARRAY[1..MAX_AXIS] OF DINT;
  _XfcDcTimeOfPosition        : ARRAY[1..MAX_AXIS] OF T_DCTIME32;

  // inputs
  _XfcTouchProbe              : Tc2_MC2_XFC.XFC_TouchProbe;
  _XfcTouchProbeEL1258        : Tc2_MC2_XFC.XFC_EL1258_TouchProbe;

  // input datatypes
  _XfcTouchProbeOptions       : Tc2_MC2_XFC.ST_XfcTouchProbeOptions;
  _XfcTriggerRef              : Tc2_MC2_XFC.XFC_TRIGGER_REF;
  _XfcTriggerRef_MT           : Tc2_MC2_XFC.XFC_MT_TRIGGER_REF;      // multi timestamping
  //_XfcEl1258Interface_MT      : Tc2_MC2_XFC.EL1258_MT_IoInterface;   // multi timestamping
  _XfcRecordedPosition_MT     : Tc2_MC2_XFC.ST_RecordedPosition;     // multi timestamping


  // outputs
  _XfcOutputEL2252            : Tc2_MC2_XFC.XFC_TouchProbe;
  _XfcOutputEL2258            : Tc2_MC2_XFC.XFC_EL2258_MultiEdge;

 
  // work vars

END_VAR

METHOD Check : BOOL
VAR_INST
  _idx        : UINT;
  _eCheck     : E_XFC_CHECK;
END_VAR

FOR _idx := 1 TO MAX_AXIS
DO
  IF NOT (_ItfAxis[_idx] <> 0)
  THEN
    _eCheck       := E_XFC_CHECK.XFC_CHECK_REF_AXIS_ITF;
    RETURN;
  END_IF
END_FOR




_eCheck           := E_XFC_CHECK.XFC_CHECK_DONE;
Check             := TRUE;
END_METHOD

//-----------------------------------------------------------------------------------------------------------
// GetIndex
//
// HAUD
// 18.07.2024
// - input:  TwinCAT NC Axis ID
// - output: index in AXIS_REF array
//-----------------------------------------------------------------------------------------------------------
METHOD GetIndex : UDINT
VAR_INPUT
  AxisId        : UDINT;
END_VAR
VAR
  _idx          : UDINT;
END_VAR

FOR _idx := 1 TO TO_UDINT(MAX_AXIS)
DO
  IF (_ItfAxis[_idx].AxisRef.NcToPlc.AxisId > 0)
  THEN
    IF (_ItfAxis[_idx].AxisRef.NcToPlc.AxisId = AxisId)
    THEN
      GetIndex      := _idx;
      RETURN;
    END_IF
  END_IF
END_FOR

GetIndex          := _idx;
END_METHOD

PROPERTY ItfAxis : ARRAY[1..MAX_AXIS]       OF I_McAxis
SET
_ItfAxis := ItfAxis;
END_SET
END_PROPERTY

METHOD PositionAtTime : E_PROGRESS
VAR_INPUT
  Execute         : BOOL;
  AxisId          : UDINT;                    // NC Axis ID
  DcTime          : Tc2_EtherCAT.T_DCTIME32;  // lower part Dctime of event
  MessageLevel    : E_MessageType := E_MessageType.eMessageError;  // switch for detailed logging if required
END_VAR
VAR_INST
  _eState         : E_PROGRESS;

  _stMsg          : ST_Message;
  _bError         : BOOL;
  _udiErrorId     : UDINT;
  _AxisIndex      : UDINT;
END_VAR
IF NOT Execute THEN _eState     := E_PROGRESS.PROGRESS_INIT;  END_IF
IF NOT Check() THEN PositionAtTime   := E_PROGRESS.PROGRESS_ERROR; END_IF

CASE _eState
OF
  E_PROGRESS.PROGRESS_INIT:
    IF Execute
    THEN
      _AxisIndex                := GetIndex(AxisId);
      _bError                   := FALSE;
      _udiErrorId               := 0;
      _eState                   := E_PROGRESS.PROGRESS_BUSY;

      IF (MessageLevel = E_MessageType.eMessageVerbose)
      THEN
        _stMsg.eType            := E_MessageType.eMessageVerbose;
        _stMsg.eDevice          := _eDeviceAxis;
        _stMsg.eSubdevice       := XfcPositionAtTime;
        _stMsg.iErrorNumber     := 0;
        _stMsg.sText            := TO_STRING(_eState);

        f_MessageSet(_stMsg);
      END_IF

      IF NOT (_AxisIndex > 0)
      THEN
        _stMsg.eType            := E_MessageType.eMessageError;
        _stMsg.eDevice          := _eDeviceAxis;
        _stMsg.eSubdevice       := XfcPositionAtTime;
        _stMsg.iErrorNumber     := _AxisIndex;
        _stMsg.sText            := TO_STRING(E_XFC_CHECK.XFC_CHECK_AXIS_INDEX);

        _bError                 := TRUE;
        _eState                 := E_PROGRESS.PROGRESS_STILL_WORKING;
      END_IF
    END_IF
END_CASE
//-----------------------------------------------------------------------------
//-----------------------------------------------------------------------------
CASE _eState
OF
  E_PROGRESS.PROGRESS_BUSY:
    _eState                     := E_PROGRESS.PROGRESS_STILL_WORKING;

    _XfcPositionAtTime[_AxisIndex](
                    DcTime      := DcTime, 
                    Options     := _XfcNcTimeConversionOptions[_AxisIndex], 
                    Position    => _XfcRecordedPosition[_AxisIndex], 
                    Error       => _bError, 
                    ErrorID     => _udiErrorId, 
                    Axis        := _ItfAxis[_AxisIndex].AxisRef);
END_CASE
//-----------------------------------------------------------------------------
//-----------------------------------------------------------------------------
CASE _eState
OF
  E_PROGRESS.PROGRESS_STILL_WORKING:
    IF NOT _bError
    THEN
      _eState                   := E_PROGRESS.PROGRESS_DONE;
      IF (MessageLevel > E_MessageType.eMessageWarning)
      THEN
        _stMsg.eType            := E_MessageType.eMessageInfo;
        _stMsg.eDevice          := _eDeviceAxis;
        _stMsg.eSubdevice       := XfcPositionAtTime;
        _stMsg.iErrorNumber     := 0;
        _stMsg.sText            := TO_STRING(_eState);

        f_MessageSet(_stMsg);
      END_IF
    ELSE
      _eState                   := E_PROGRESS.PROGRESS_ERROR;

      _stMsg.eType              := E_MessageType.eMessageError;
      _stMsg.eDevice            := _eDeviceAxis;
      _stMsg.eSubdevice         := XfcPositionAtTime;
      _stMsg.iErrorNumber       := _udiErrorId;
      _stMsg.sText              := TO_STRING(_eState);

      f_MessageSet(_stMsg);
    END_IF
END_CASE



PositionAtTime                  := _eState;
END_METHOD

METHOD TimeOfPosition : E_PROGRESS
VAR_INPUT
  Execute         : BOOL;
  AxisId          : UDINT;                    // NC Axis ID
  Position        : LREAL;
  MessageLevel    : E_MessageType := E_MessageType.eMessageError;  // switch for detailed logging if required
END_VAR
VAR_INST
  _eState         : E_PROGRESS;

  _stMsg          : ST_Message;
  _bError         : BOOL;
  _udiErrorId     : UDINT;
  _AxisIndex      : UDINT;
END_VAR
IF NOT Execute THEN _eState     := E_PROGRESS.PROGRESS_INIT;  END_IF
IF NOT Check() THEN TimeOfPosition   := E_PROGRESS.PROGRESS_ERROR; END_IF

CASE _eState
OF
  E_PROGRESS.PROGRESS_INIT:
    IF Execute
    THEN
      _AxisIndex                := GetIndex(AxisId);
      _bError                   := FALSE;
      _udiErrorId               := 0;
      _eState                   := E_PROGRESS.PROGRESS_BUSY;

      IF (MessageLevel = E_MessageType.eMessageVerbose)
      THEN
        _stMsg.eType            := E_MessageType.eMessageVerbose;
        _stMsg.eDevice          := _eDeviceAxis;
        _stMsg.eSubdevice       := XfcTimeOfPosition;
        _stMsg.iErrorNumber     := 0;
        _stMsg.sText            := TO_STRING(_eState);

        f_MessageSet(_stMsg);
      END_IF

      IF NOT (_AxisIndex > 0)
      THEN
        _stMsg.eType            := E_MessageType.eMessageError;
        _stMsg.eDevice          := _eDeviceAxis;
        _stMsg.eSubdevice       := XfcTimeOfPosition;
        _stMsg.iErrorNumber     := _AxisIndex;
        _stMsg.sText            := TO_STRING(E_XFC_CHECK.XFC_CHECK_AXIS_INDEX);

        _bError                 := TRUE;
        _eState                 := E_PROGRESS.PROGRESS_STILL_WORKING;
      END_IF
    END_IF
END_CASE
//-----------------------------------------------------------------------------
//-----------------------------------------------------------------------------
CASE _eState
OF
  E_PROGRESS.PROGRESS_BUSY:
    _eState                     := E_PROGRESS.PROGRESS_STILL_WORKING;

    _XfcTimeOfPosition[_AxisIndex](
	                  Position    := Position, 
                    Options     := _XfcNcTimeConversionOptions[_AxisIndex], 
                    DcTime      => _XfcRecordedTime[_AxisIndex], 
                    Error       => _bError, 
                    ErrorID     => _udiErrorId, 
                    Axis        := _ItfAxis[_AxisIndex].AxisRef);
END_CASE
//-----------------------------------------------------------------------------
//-----------------------------------------------------------------------------
CASE _eState
OF
  E_PROGRESS.PROGRESS_STILL_WORKING:
    IF NOT _bError
    THEN
      _eState                   := E_PROGRESS.PROGRESS_DONE;
      IF (MessageLevel > E_MessageType.eMessageWarning)
      THEN
        _stMsg.eType            := E_MessageType.eMessageInfo;
        _stMsg.eDevice          := _eDeviceAxis;
        _stMsg.eSubdevice       := XfcTimeOfPosition;
        _stMsg.iErrorNumber     := 0;
        _stMsg.sText            := TO_STRING(_eState);

        f_MessageSet(_stMsg);
      END_IF
    ELSE
      _eState                   := E_PROGRESS.PROGRESS_ERROR;

      _stMsg.eType              := E_MessageType.eMessageError;
      _stMsg.eDevice            := _eDeviceAxis;
      _stMsg.eSubdevice         := XfcTimeOfPosition;
      _stMsg.iErrorNumber       := _udiErrorId;
      _stMsg.sText              := TO_STRING(_eState);

      f_MessageSet(_stMsg);
    END_IF
END_CASE



TimeOfPosition                  := _eState;
END_METHOD

METHOD TimeToPosition : E_PROGRESS
VAR_INPUT
  Execute         : BOOL;
  AxisId          : UDINT;                    // NC Axis ID
  TargetPosition  : LREAL;
  MessageLevel    : E_MessageType := E_MessageType.eMessageError;  // switch for detailed logging if required
END_VAR
VAR_INST
  _eState         : E_PROGRESS;

  _stMsg          : ST_Message;
  _bError         : BOOL;
  _udiErrorId     : UDINT;
  _AxisIndex      : UDINT;
END_VAR
IF NOT Execute THEN _eState     := E_PROGRESS.PROGRESS_INIT;  END_IF
IF NOT Check() THEN TimeToPosition   := E_PROGRESS.PROGRESS_ERROR; END_IF

CASE _eState
OF
  E_PROGRESS.PROGRESS_INIT:
    IF Execute
    THEN
      _AxisIndex                := GetIndex(AxisId);
      _bError                   := FALSE;
      _udiErrorId               := 0;
      _eState                   := E_PROGRESS.PROGRESS_BUSY;

      IF (MessageLevel = E_MessageType.eMessageVerbose)
      THEN
        _stMsg.eType            := E_MessageType.eMessageVerbose;
        _stMsg.eDevice          := _eDeviceAxis;
        _stMsg.eSubdevice       := XfcTimeToPosition;
        _stMsg.iErrorNumber     := 0;
        _stMsg.sText            := TO_STRING(_eState);

        f_MessageSet(_stMsg);
      END_IF

      IF NOT (_AxisIndex > 0)
      THEN
        _stMsg.eType            := E_MessageType.eMessageError;
        _stMsg.eDevice          := _eDeviceAxis;
        _stMsg.eSubdevice       := XfcTimeToPosition;
        _stMsg.iErrorNumber     := _AxisIndex;
        _stMsg.sText            := TO_STRING(E_XFC_CHECK.XFC_CHECK_AXIS_INDEX);

        _bError                 := TRUE;
        _eState                 := E_PROGRESS.PROGRESS_STILL_WORKING;
      END_IF
    END_IF
END_CASE
//-----------------------------------------------------------------------------
//-----------------------------------------------------------------------------
CASE _eState
OF
  E_PROGRESS.PROGRESS_BUSY:
    _eState                     := E_PROGRESS.PROGRESS_STILL_WORKING;

    _XfcTimeToPosition[_AxisIndex](
                Position        := TargetPosition, 
                Options         := _XfcNcTimeConversionOptions[_AxisIndex], 
                Duration        => _XfcDurationToPosition[_AxisIndex], 
                TimeOfPosition  => _XfcDcTimeOfPosition[_AxisIndex], 
                Error           => _bError, 
                ErrorID         => _udiErrorId, 
                Axis            := _ItfAxis[_AxisIndex].AxisRef);
END_CASE
//-----------------------------------------------------------------------------
//-----------------------------------------------------------------------------
CASE _eState
OF
  E_PROGRESS.PROGRESS_STILL_WORKING:
    IF NOT _bError
    THEN
      _eState                   := E_PROGRESS.PROGRESS_DONE;
      IF (MessageLevel > E_MessageType.eMessageWarning)
      THEN
        _stMsg.eType            := E_MessageType.eMessageInfo;
        _stMsg.eDevice          := _eDeviceAxis;
        _stMsg.eSubdevice       := XfcTimeToPosition;
        _stMsg.iErrorNumber     := 0;
        _stMsg.sText            := TO_STRING(_eState);

        f_MessageSet(_stMsg);
      END_IF
    ELSE
      _eState                   := E_PROGRESS.PROGRESS_ERROR;

      _stMsg.eType              := E_MessageType.eMessageError;
      _stMsg.eDevice            := _eDeviceAxis;
      _stMsg.eSubdevice         := XfcTimeToPosition;
      _stMsg.iErrorNumber       := _udiErrorId;
      _stMsg.sText              := TO_STRING(_eState);

      f_MessageSet(_stMsg);
    END_IF
END_CASE



TimeToPosition                  := _eState;
END_METHOD

METHOD TimeToPositionModulo : E_PROGRESS
VAR_INPUT
  Execute         : BOOL;
  AxisId          : UDINT;                    // NC Axis ID
  ModuloPosition  : LREAL;
  ModuloFactor    : LREAL;
  MessageLevel    : E_MessageType := E_MessageType.eMessageError;  // switch for detailed logging if required
END_VAR
VAR_INST
  _eState         : E_PROGRESS;

  _stMsg          : ST_Message;
  _bError         : BOOL;
  _udiErrorId     : UDINT;
  _AxisIndex      : UDINT;
END_VAR
IF NOT Execute THEN _eState     := E_PROGRESS.PROGRESS_INIT;  END_IF
IF NOT Check() THEN TimeToPositionModulo   := E_PROGRESS.PROGRESS_ERROR; END_IF

CASE _eState
OF
  E_PROGRESS.PROGRESS_INIT:
    IF Execute
    THEN
      _AxisIndex                := GetIndex(AxisId);
      _bError                   := FALSE;
      _udiErrorId               := 0;
      _eState                   := E_PROGRESS.PROGRESS_BUSY;

      IF (MessageLevel = E_MessageType.eMessageVerbose)
      THEN
        _stMsg.eType            := E_MessageType.eMessageVerbose;
        _stMsg.eDevice          := _eDeviceAxis;
        _stMsg.eSubdevice       := XfcTimeToModuloPosition;
        _stMsg.iErrorNumber     := 0;
        _stMsg.sText            := TO_STRING(_eState);

        f_MessageSet(_stMsg);
      END_IF

      IF NOT (_AxisIndex > 0)
      THEN
        _stMsg.eType            := E_MessageType.eMessageError;
        _stMsg.eDevice          := _eDeviceAxis;
        _stMsg.eSubdevice       := XfcTimeToModuloPosition;
        _stMsg.iErrorNumber     := _AxisIndex;
        _stMsg.sText            := TO_STRING(E_XFC_CHECK.XFC_CHECK_AXIS_INDEX);

        _bError                 := TRUE;
        _eState                 := E_PROGRESS.PROGRESS_STILL_WORKING;
      END_IF
    END_IF
END_CASE
//-----------------------------------------------------------------------------
//-----------------------------------------------------------------------------
CASE _eState
OF
  E_PROGRESS.PROGRESS_BUSY:
    _eState                     := E_PROGRESS.PROGRESS_STILL_WORKING;

    _XfcTimeToModuloPosition[_AxisIndex](
                Position        := ModuloPosition, 
                ModuloFactor    := ModuloFactor, 
                Options         := _XfcNcTimeConversionOptions[_AxisIndex], 
                Duration        => _XfcDurationToPosition[_AxisIndex], 
                AbsolutePosition=> _XfcRecordedPosition[_AxisIndex], 
                TimeOfPosition  => _XfcDcTimeOfPosition[_AxisIndex], 
                Error           => _bError, 
                ErrorID         => _udiErrorId, 
                Axis            := _ItfAxis[_AxisIndex].AxisRef);
END_CASE
//-----------------------------------------------------------------------------
//-----------------------------------------------------------------------------
CASE _eState
OF
  E_PROGRESS.PROGRESS_STILL_WORKING:
    IF NOT _bError
    THEN
      _eState                   := E_PROGRESS.PROGRESS_DONE;
      IF (MessageLevel > E_MessageType.eMessageWarning)
      THEN
        _stMsg.eType            := E_MessageType.eMessageInfo;
        _stMsg.eDevice          := _eDeviceAxis;
        _stMsg.eSubdevice       := XfcTimeToModuloPosition;
        _stMsg.iErrorNumber     := 0;
        _stMsg.sText            := TO_STRING(_eState);

        f_MessageSet(_stMsg);
      END_IF
    ELSE
      _eState                   := E_PROGRESS.PROGRESS_ERROR;

      _stMsg.eType              := E_MessageType.eMessageError;
      _stMsg.eDevice            := _eDeviceAxis;
      _stMsg.eSubdevice         := XfcTimeToModuloPosition;
      _stMsg.iErrorNumber       := _udiErrorId;
      _stMsg.sText              := TO_STRING(_eState);

      f_MessageSet(_stMsg);
    END_IF
END_CASE

TimeToPositionModulo                  := _eState;
END_METHOD

METHOD WaitForPosition : E_PROGRESS
VAR_INPUT
  Execute         : BOOL;
  AxisId          : UDINT;                    // NC Axis ID
  TargetPosition  : LREAL;
  MessageLevel    : E_MessageType := E_MessageType.eMessageError;  // switch for detailed logging if required
END_VAR
VAR_INST
  _eState         : E_PROGRESS;

  _stMsg          : ST_Message;
  _bError         : BOOL;
  _udiErrorId     : UDINT;
  _AxisIndex      : UDINT;
END_VAR
IF NOT Execute THEN _eState     := E_PROGRESS.PROGRESS_INIT;  END_IF
IF NOT Check() THEN WaitForPosition   := E_PROGRESS.PROGRESS_ERROR; END_IF

CASE _eState
OF
  E_PROGRESS.PROGRESS_INIT:
    IF Execute
    THEN
      _AxisIndex                := GetIndex(AxisId);
      _bError                   := FALSE;
      _udiErrorId               := 0;
      _eState                   := E_PROGRESS.PROGRESS_BUSY;

      IF (MessageLevel = E_MessageType.eMessageVerbose)
      THEN
        _stMsg.eType            := E_MessageType.eMessageVerbose;
        _stMsg.eDevice          := _eDeviceAxis;
        _stMsg.eSubdevice       := XfcWaitForPosition;
        _stMsg.iErrorNumber     := 0;
        _stMsg.sText            := TO_STRING(_eState);

        f_MessageSet(_stMsg);
      END_IF

      IF NOT (_AxisIndex > 0)
      THEN
        _stMsg.eType            := E_MessageType.eMessageError;
        _stMsg.eDevice          := _eDeviceAxis;
        _stMsg.eSubdevice       := XfcWaitForPosition;
        _stMsg.iErrorNumber     := _AxisIndex;
        _stMsg.sText            := TO_STRING(E_XFC_CHECK.XFC_CHECK_AXIS_INDEX);

        _bError                 := TRUE;
        _eState                 := E_PROGRESS.PROGRESS_STILL_WORKING;
      END_IF
    END_IF
END_CASE
//-----------------------------------------------------------------------------
//-----------------------------------------------------------------------------
CASE _eState
OF
  E_PROGRESS.PROGRESS_BUSY:
    _eState                     := E_PROGRESS.PROGRESS_PREPARE;

    _XfcTimeToPosition[_AxisIndex](
                Position        := TargetPosition, 
                Options         := _XfcNcTimeConversionOptions[_AxisIndex], 
                Duration        => _XfcDurationToPosition[_AxisIndex], 
                TimeOfPosition  => , 
                Error           => _bError, 
                ErrorID         => _udiErrorId, 
                Axis            := _ItfAxis[_AxisIndex].AxisRef);

END_CASE
//-----------------------------------------------------------------------------
//-----------------------------------------------------------------------------
CASE _eState
OF
  E_PROGRESS.PROGRESS_PREPARE:

    IF NOT _bError
    THEN
      IF (_XfcTimeToPosition[_AxisIndex].Duration < 10_000_000)
      THEN
        _eState                 := E_PROGRESS.PROGRESS_STILL_WORKING;
      ELSE
        _eState                 := E_PROGRESS.PROGRESS_BUSY;
      END_IF
    ELSE
      IF (_udiErrorId <> 17250)
      THEN
        // axis is not yet in range --> retry
        _eState                 := E_PROGRESS.PROGRESS_BUSY;
      ELSE
        // position will not be reachable --> error
        _eState                 := E_PROGRESS.PROGRESS_STILL_WORKING;  
      END_IF
    END_IF
END_CASE
//-----------------------------------------------------------------------------
//-----------------------------------------------------------------------------
CASE _eState
OF
  E_PROGRESS.PROGRESS_STILL_WORKING:
    IF NOT _bError
    THEN
      _eState                   := E_PROGRESS.PROGRESS_DONE;
      IF (MessageLevel > E_MessageType.eMessageWarning)
      THEN
        _stMsg.eType            := E_MessageType.eMessageInfo;
        _stMsg.eDevice          := _eDeviceAxis;
        _stMsg.eSubdevice       := XfcWaitForPosition;
        _stMsg.iErrorNumber     := TO_ULINT(_XfcDurationToPosition[_AxisIndex]);
        _stMsg.sText            := TO_STRING(_eState);

        f_MessageSet(_stMsg);
      END_IF
    ELSE
      _eState                   := E_PROGRESS.PROGRESS_ERROR;

      _stMsg.eType              := E_MessageType.eMessageError;
      _stMsg.eDevice            := _eDeviceAxis;
      _stMsg.eSubdevice         := XfcWaitForPosition;
      _stMsg.iErrorNumber       := _udiErrorId;
      _stMsg.sText              := TO_STRING(_eState);

      f_MessageSet(_stMsg);
    END_IF
END_CASE


WaitForPosition                 := _eState;
END_METHOD

END_FUNCTION_BLOCK

// ---- PLC_MOTION/NC_PTP/class/FB_McAxisCtrl.TcPOU
FUNCTION_BLOCK FB_McAxisCtrl EXTENDS FB_McAxisBase
VAR
  _eCheck                   : E_CHECK_STATE;  // pointer check

  _eAxisCycle,                                // cyclic AXIS_REF() and MC_Power check
  _eInit                    : E_PROGRESS;     // axis startup and init, get encoder type, get axis name, get device name

  _nAxisIndex               : UINT;           // know thyself
  _rTargetWindow            : LREAL := 0.1;   // TODO: get that from NC

  // access to CoE register for hardware device name
  _sDeviceName              : STRING(256) := 'NO NAME';
  _fbCoeRead				        : Tc2_MC2_Drive.FB_CoERead;

  // pointers to all; access required for coupling; access by index
  _Axes                     : REFERENCE TO ARRAY[1..PLC_CONSTANT.MAX_AXIS] OF AXIS_REF;

  _Ctrl                     : POINTER TO ARRAY[1..PLC_CONSTANT.MAX_AXIS] OF ST_AXIS_CTRL;    // contains command to be executed
  _State                    : POINTER TO ARRAY[1..PLC_CONSTANT.MAX_AXIS] OF ST_AXIS_STATE;   // mirrors command with added result

  _Info                     : POINTER TO ARRAY[1..PLC_CONSTANT.MAX_AXIS] OF ST_AXIS_INFO;    // axis state and position data to read from
  _Data                     : POINTER TO ARRAY[1..PLC_CONSTANT.MAX_AXIS] OF ST_AXIS_MOVE_DATA;    // structure for cyclic interface

  _NcParameterIn            : POINTER TO ARRAY[1..PLC_CONSTANT.MAX_AXIS] OF ST_NC_PARAMETER; // W struct for a single parameter
  _NcParameterOut           : POINTER TO ARRAY[1..PLC_CONSTANT.MAX_AXIS] OF ST_NC_PARAMETER; // R struct for a single parameter
  _HomeParameter            : POINTER TO ARRAY[1..PLC_CONSTANT.MAX_AXIS] OF ST_HOMING;       // homing parameter for each axis

  _GearInParameter          : POINTER TO ARRAY[1..PLC_CONSTANT.MAX_AXIS] OF ST_GEAR_IN;      // Master Indices, dyn constraints for simple GearIn

  _MotionOptions            : POINTER TO ARRAY[1..PLC_CONSTANT.MAX_AXIS] OF ST_MOTION_OPTIONS;

  _LimitSwitches            : POINTER TO ARRAY[1..PLC_CONSTANT.MAX_AXIS] OF ST_AXIS_LIMIT_SWITCHES;

  // local copies of command
  _eCmd,
  _eCmdOld                       : E_AXIS_CTRL;

  // Last handled NC Axis parameter to write
  _eParameterNrWrite              : Tc2_MC2.MC_AxisParameter;
  _rParameterWrtValue             : LREAL;

  // Last handled NC Axis parameter to read
  _eParameterNrRead               : Tc2_MC2.MC_AxisParameter;
  _rParameterReadValue            : LREAL;

  // execution state
  _eResult                        : E_PROGRESS;   // result of execution state
  _eResultOld                     : E_PROGRESS;   // old result for detecting change
  _eState                         : E_AXIS_STATE; // execution state

  // calibration options with limit switches and simulation
  _bCalibrationCam                : BOOL;

  // placeholder dummies in case count of Multimaster ases <> 4
  {attribute 'hide'}
  _MultiMasterDummyRef            : ARRAY[1..4] OF AXIS_REF;

  _fbGearOut                      : Tc2_MC2.MC_GearOut;
  _fbGearIn                       : Tc2_MC2.MC_GearIn;
  _fbGearInMultiMaster            : Tc2_MC2.MC_GearInMultiMaster;
END_VAR

IF NOT Check() THEN RETURN; END_IF
//-----------------------------------------------------------------------------
// check _HomeParameter for calibration input options
//-----------------------------------------------------------------------------
_bCalibrationCam                    := GetCalibrationCam();
CalibrationCam                      := ADR(_bCalibrationCam);
//-----------------------------------------------------------------------------
//-----------------------------------------------------------------------------
Override                            := _Data^[_nAxisIndex].rOverride;
//-----------------------------------------------------------------------------
//-----------------------------------------------------------------------------
// cyclic call to MC_Power and AXIS_REF()
//-----------------------------------------------------------------------------
_eAxisCycle                         := Cycle();
//-----------------------------------------------------------------------------
//-----------------------------------------------------------------------------
// get command from outside world
//-----------------------------------------------------------------------------
_eCmd                               := _Ctrl^[_nAxisIndex].eCmd;
//-----------------------------------------------------------------------------
//-----------------------------------------------------------------------------
//  OnChange react to command
//-----------------------------------------------------------------------------
IF (_eCmd <> _eCmdOld)
THEN
  // get busy
  _eState                           := Cmd(_eCmd); // get execution state for command
  _eCmdOld                          := _eCmd;
  LogControl();
END_IF
//-----------------------------------------------------------------------------
//-----------------------------------------------------------------------------
// Check AxisInit
//-----------------------------------------------------------------------------
IF NOT (_eInit = E_PROGRESS.PROGRESS_DONE)
THEN
  _Info^[_nAxisIndex].bReady        := FALSE;
ELSE
  _Info^[_nAxisIndex].bReady        := _AxisRef.Status.ControlLoopClosed AND
                                       (NOT _AxisRef.Status.Error)       AND 
                                       (NOT _AxisRef.Status.Moving);
END_IF
//-----------------------------------------------------------------------------
//-----------------------------------------------------------------------------
//  execution result
//-----------------------------------------------------------------------------
CASE _eResult
OF
  E_PROGRESS.PROGRESS_INVALID:
    _State^[_nAxisIndex].eState     := TO_UINT(E_PROGRESS.PROGRESS_ERROR);

  E_PROGRESS.PROGRESS_ERROR:
    _Info^[_nAxisIndex].bReady      := FALSE;
    _Info^[_nAxisIndex].bError      := TRUE;
    _Info^[_nAxisIndex].nErrorId    := ErrorId;

    _State^[_nAxisIndex].eState     := _eState + E_PROGRESS.PROGRESS_ERROR;

  E_PROGRESS.PROGRESS_DONE:
    _State^[_nAxisIndex].eState     := _eState + E_PROGRESS.PROGRESS_DONE;

ELSE
  //-----------------------------------------------------------------------------
  // execution state result to interface
  //-----------------------------------------------------------------------------
  _State^[_nAxisIndex].eState       := _eState + _eResult;

  //-----------------------------------------------------------------------------
  //-----------------------------------------------------------------------------
  //  execution state for command
  //-----------------------------------------------------------------------------
  CASE _eState
  OF
    E_AXIS_STATE.AXIS_INIT:
      //-------------------------------------------------------------------------
      // axis always requires one init from outside world at startup
      // _eInit has to be valid for other commands to be accepted in Cmd(_eCtrl)
      _eInit := _eResult            := AxisInit(TRUE);
  
    E_AXIS_STATE.AXIS_NO_INIT:
      //-------------------------------------------------------------------------
      // we are here because you sent a command before having done AXIS_INIT
      _eResult                      := E_PROGRESS.PROGRESS_ERROR;
  
    E_AXIS_STATE.AXIS_DISABLE:
      _eResult                      := AxisDisable(TRUE);
  
    E_AXIS_STATE.AXIS_ENABLE:
      _eResult                      := AxisEnable(TRUE);
  
    E_AXIS_STATE.AXIS_IDLE:
      _eResult                      := AxisIdle(TRUE);
  
    E_AXIS_STATE.AXIS_HOME:
      _eResult                      := AxisHome(TRUE);
  
    E_AXIS_STATE.AXIS_MOVE_POS:
      _eResult                      := AxisMoveToPosition(TRUE, _Data^[_nAxisIndex]);
  
    E_AXIS_STATE.AXIS_MOVE_VELO:
      _eResult                      := AxisMoveVelocity(TRUE, _Data^[_nAxisIndex]);

    E_AXIS_STATE.AXIS_SEND_TO_POS:
      _eResult                      := AxisSendToPosition(TRUE, _Data^[_nAxisIndex]);
  
    E_AXIS_STATE.AXIS_RESET:
      _eResult                      := AxisReset(TRUE);
  
    E_AXIS_STATE.AXIS_HALT:
      _eResult                      := AxisHalt(TRUE, _Data^[_nAxisIndex]);
  
    E_AXIS_STATE.AXIS_STOP:
      _eResult                      := AxisStop(TRUE, _Data^[_nAxisIndex]);
  
    E_AXIS_STATE.AXIS_MOVE_BUFFER:
      _eResult                      := AxisBufferPos(TRUE, _Data^[_nAxisIndex]);
  
    E_AXIS_STATE.AXIS_MOVE_BUFFER_VELO:
      _eResult                      := AxisBufferVelo(TRUE, _Data^[_nAxisIndex]);
  
    E_AXIS_STATE.AXIS_PARAMETER_READ:
      _eResult                      := AxisParameterRead(TRUE, _eParameterNrRead);

    E_AXIS_STATE.AXIS_PARAMETER_WRITE:
      _eResult                      := AxisParameterWrite(TRUE, _eParameterNrWrite);
  
    E_AXIS_STATE.AXIS_PARAMETER_WRITE_PERSISTENT:
      _eResult                      := AxisParameterWritePersistent(FALSE, _eParameterNrWrite);
  
    E_AXIS_STATE.AXIS_GEAR_IN:
      _eResult                      := AxisGearIn(TRUE);
  
    E_AXIS_STATE.AXIS_GEAR_OUT:
      _eResult                      := AxisGearOut(TRUE);
  
    E_AXIS_STATE.AXIS_GEAR_IN_MULTIMASTER:
      _eResult                      := AxisGearInMultiMaster(TRUE);
  
  ELSE
    IF (_eCmd > E_AXIS_CTRL.AXIS_NULL)
    THEN
      _eResult                      := E_PROGRESS.PROGRESS_NOT_EXIST;
      _Info^[_nAxisIndex].bError    := TRUE;
    ELSE
      _eResult                      := E_PROGRESS.PROGRESS_INVALID;
    END_IF
  END_CASE
END_CASE
//-----------------------------------------------------------------------------
//-----------------------------------------------------------------------------
//  OnChange of execution state result
//    - log result and clear error number on interface
//-----------------------------------------------------------------------------
IF (_eResult <> _eResultOld)
THEN
  LogResult();
  _Info^[_nAxisIndex].nErrorId      := 0;
  _eResultOld                       := _eResult;
END_IF
//-----------------------------------------------------------------------------
// encoder type (enum)
//-----------------------------------------------------------------------------
_State^[_nAxisIndex].eAxisEncoder   := EncoderType;
//-----------------------------------------------------------------------------
// Check ControlLoop
//-----------------------------------------------------------------------------
IF _AxisRef.Status.ControlLoopClosed
THEN
  _Info^[_nAxisIndex].bEnabled      := TRUE;
ELSE
  _Info^[_nAxisIndex].bEnabled      := FALSE;
END_IF
//-----------------------------------------------------------------------------
_Info^[_nAxisIndex].bStandstill     := _AxisRef.Status.NotMoving;
//-----------------------------------------------------------------------------
_Info^[_nAxisIndex].rActPos         := _AxisRef.NcToPlc.ActPos;
_Info^[_nAxisIndex].rActVelo        := _AxisRef.NcToPlc.ActVelo;
_Info^[_nAxisIndex].rPosDiff        := _AxisRef.NcToPlc.PosDiff;
//-----------------------------------------------------------------------------
IF (_Info^[_nAxisIndex].rActPos < _Data^[_nAxisIndex].rSetPos + _rTargetWindow) AND
   (_Info^[_nAxisIndex].rActPos > _Data^[_nAxisIndex].rSetPos - _rTargetWindow) AND
    _Info^[_nAxisIndex].bStandstill
THEN
  _Info^[_nAxisIndex].bInTarget     := TRUE;
ELSE
  _Info^[_nAxisIndex].bInTarget     := FALSE;
END_IF
//-----------------------------------------------------------------------------
// copy CoupleState from axis
//-----------------------------------------------------------------------------
_Info^[_nAxisIndex].dwCoupleState   := _AxisRef.NcToPlc.CoupleState;
//-----------------------------------------------------------------------------
//-----------------------------------------------------------------------------
// copy NC AxisId from axis
//-----------------------------------------------------------------------------
_Info^[_nAxisIndex].nNcAxisId       := _AxisRef.NcToPlc.AxisId;
//-----------------------------------------------------------------------------

PROPERTY Axes : reference TO ARRAY[1..PLC_CONSTANT.MAX_AXIS] OF AXIS_REF
SET
_Axes REF= Axes;
END_SET
END_PROPERTY

METHOD AxisBufferPos : E_PROGRESS
VAR_INPUT
  bEnable            : BOOL;
  Data              : ST_AXIS_MOVE_DATA;
END_VAR
VAR_INST
  _BufferMode       : Tc2_MC2.MC_BufferMode;
  _eres,
  _eState           : E_PROGRESS;
END_VAR
IF NOT Check() THEN AxisBufferPos := E_PROGRESS.PROGRESS_ERROR; RETURN; END_IF
IF NOT bEnable THEN _eState := E_PROGRESS.PROGRESS_INIT; END_IF

CASE _eState
OF
  E_PROGRESS.PROGRESS_INIT:
    IF bEnable 
    THEN
      _eState       := E_PROGRESS.PROGRESS_BUSY;
    END_IF
END_CASE
CASE _eState
OF
  E_PROGRESS.PROGRESS_BUSY:
    _eState         := E_PROGRESS.PROGRESS_WORKING;
    _BufferMode     := _MotionOptions^[_nAxisIndex].eBufferMode;
    _eres           := MovePosBuffer(
                                  bEnable      := FALSE, 
                                  Position    := Data.rSetPos, 
                                  Vel         := Data.rSetVelo, 
                                  Acc         := Data.rAcc, 
                                  Dec         := Data.rDec, 
                                  Jerk        := Data.rJerk, 
                                  BufferMode  := _BufferMode);
END_CASE
CASE _eState
OF
  E_PROGRESS.PROGRESS_WORKING:
    _BufferMode     := _MotionOptions^[_nAxisIndex].eBufferMode;
    AxisBufferPos   := _eres  
                    := MovePosBuffer(
                                  bEnable      := TRUE, 
                                  Position    := Data.rSetPos, 
                                  Vel         := Data.rSetVelo, 
                                  Acc         := Data.rAcc, 
                                  Dec         := Data.rDec, 
                                  Jerk        := Data.rJerk, 
                                  BufferMode  := _BufferMode);
    IF (_eres = E_PROGRESS.PROGRESS_ERROR)
    THEN
      _eState       := E_PROGRESS.PROGRESS_ERROR;

    ELSIF (_Ctrl^[_nAxisIndex].eProgress = E_PROGRESS.PROGRESS_DONE)
    THEN
      // when Ctrl decides to leave; make finishing move and be done
      _eState       := E_PROGRESS.PROGRESS_DONE;
    END_IF
END_CASE
CASE _eState
OF
  E_PROGRESS.PROGRESS_ERROR,
  E_PROGRESS.PROGRESS_DONE:
    _eres           := MovePosBuffer(
                                  bEnable      := FALSE, 
                                  Position    := Data.rSetPos, 
                                  Vel         := Data.rSetVelo, 
                                  Acc         := Data.rAcc, 
                                  Dec         := Data.rDec, 
                                  Jerk        := Data.rJerk, 
                                  BufferMode  := _BufferMode);

    AxisBufferPos   := _eState;
END_CASE
END_METHOD

METHOD AxisBufferVelo : E_PROGRESS
VAR_INPUT
  bEnable            : BOOL;
  Data              : ST_AXIS_MOVE_DATA;
END_VAR
VAR_INST
  _BufferMode       : Tc2_MC2.MC_BufferMode;
  _eres,
  _eState           : E_PROGRESS;
END_VAR
IF NOT Check() THEN AxisBufferVelo := E_PROGRESS.PROGRESS_ERROR; RETURN; END_IF
IF NOT bEnable THEN _eState := E_PROGRESS.PROGRESS_INIT; END_IF

CASE _eState
OF
  E_PROGRESS.PROGRESS_INIT:
    IF bEnable 
    THEN
      _eState       := E_PROGRESS.PROGRESS_BUSY;
    END_IF
END_CASE
CASE _eState
OF
  E_PROGRESS.PROGRESS_BUSY:
    _eState         := E_PROGRESS.PROGRESS_WORKING;
    _BufferMode     := _MotionOptions^[_nAxisIndex].eBufferMode;
    _eres           := MoveVeloBuffer(
                                  bEnable      := FALSE, 
                                  Velocity    := Data.rSetVelo, 
                                  Acc         := Data.rAcc, 
                                  Dec         := Data.rDec, 
                                  Jerk        := Data.rJerk, 
                                  BufferMode  := _BufferMode);

END_CASE
CASE _eState
OF
  E_PROGRESS.PROGRESS_WORKING:
    _BufferMode     := _MotionOptions^[_nAxisIndex].eBufferMode;
    _eres           := MoveVeloBuffer(
                                  bEnable      := TRUE, 
                                  Velocity    := Data.rSetVelo, 
                                  Acc         := Data.rAcc, 
                                  Dec         := Data.rDec, 
                                  Jerk        := Data.rJerk, 
                                  BufferMode  := _BufferMode);
    IF (_eres = E_PROGRESS.PROGRESS_ERROR)
    THEN
      _eState := E_PROGRESS.PROGRESS_ERROR;
                       MoveVeloBuffer(
                                  bEnable      := FALSE, 
                                  Velocity    := Data.rSetVelo, 
                                  Acc         := Data.rAcc, 
                                  Dec         := Data.rDec, 
                                  Jerk        := Data.rJerk, 
                                  BufferMode  := _BufferMode);

    ELSIF (_Ctrl^[_nAxisIndex].eProgress = E_PROGRESS.PROGRESS_DONE)
    THEN
      // when Ctrl decides to leave; make finishing move and be done
      _eState       := E_PROGRESS.PROGRESS_STILL_WORKING;
    END_IF
END_CASE
CASE _eState
OF
  E_PROGRESS.PROGRESS_STILL_WORKING:
    _eState         := E_PROGRESS.PROGRESS_DONE;
    _eres           := MoveVeloBuffer(
                                  bEnable      := FALSE, 
                                  Velocity    := Data.rSetVelo, 
                                  Acc         := Data.rAcc, 
                                  Dec         := Data.rDec, 
                                  Jerk        := Data.rJerk, 
                                  BufferMode  := _BufferMode);
END_CASE

AxisBufferVelo      := _eState;
END_METHOD

PROPERTY AxisCtrl : pointer to ARRAY[1..PLC_CONSTANT.MAX_AXIS] OF st_axis_ctrl
SET
_Ctrl := AxisCtrl;
END_SET
END_PROPERTY

PROPERTY AxisData : pointer to ARRAY[1..PLC_CONSTANT.MAX_AXIS] OF ST_AXIS_MOVE_DATA
SET
_Data := AxisData;
END_SET
END_PROPERTY

METHOD AxisDisable : E_PROGRESS
VAR_INPUT
  Execute           : BOOL;
END_VAR
VAR_INST
  _eState,
  _eResult          : E_PROGRESS;
  _rValue           : LREAL;
  _udiErr           : UDINT;
  _stMsg            : ST_Message;


END_VAR
IF NOT Check() THEN AxisDisable := E_PROGRESS.PROGRESS_ERROR; RETURN; END_IF
IF NOT Execute THEN _eState := E_PROGRESS.PROGRESS_INIT; END_IF

CASE _eState
OF
  E_PROGRESS.PROGRESS_INIT:
    IF Execute 
    THEN
      memset(ADR(_stMsg),0,SIZEOF(_stMsg));
      _udiErr                       := 0;
      _rValue                       := 0;
      _eState                       := E_PROGRESS.PROGRESS_BUSY;
    END_IF
END_CASE
CASE _eState
OF
  E_PROGRESS.PROGRESS_BUSY:
    _eResult                        := Disable(FALSE);
    _eState                         := E_PROGRESS.PROGRESS_OCCUPIED;
END_CASE
CASE _eState
OF
  E_PROGRESS.PROGRESS_OCCUPIED:
    _eResult                        := Disable(TRUE);

    IF (_eResult = E_PROGRESS.PROGRESS_DONE)
    THEN
      _eState                       := E_PROGRESS.PROGRESS_WORKING;
    END_IF
END_CASE
CASE _eState
OF
  E_PROGRESS.PROGRESS_WORKING:
    _eState                         := E_PROGRESS.PROGRESS_DONE;
END_CASE

AxisDisable := _eState;
END_METHOD

METHOD AxisEnable : E_PROGRESS
VAR_INPUT
  Execute           : BOOL;
END_VAR
VAR_INST
  _eState,
  _eResult          : E_PROGRESS;
  _rValue           : LREAL;
  _udiErr           : UDINT;
  _stMsg            : ST_Message;


END_VAR
IF NOT Check() THEN AxisEnable := E_PROGRESS.PROGRESS_ERROR; RETURN; END_IF
IF NOT Execute THEN _eState := E_PROGRESS.PROGRESS_INIT; END_IF

CASE _eState
OF
  E_PROGRESS.PROGRESS_INIT:
    IF Execute 
    THEN
      memset(ADR(_stMsg),0,SIZEOF(_stMsg));
      _udiErr                       := 0;
      _rValue                       := 0;
      _eState                       := E_PROGRESS.PROGRESS_BUSY;
    END_IF
END_CASE
CASE _eState
OF
  E_PROGRESS.PROGRESS_BUSY:
    _eResult                        := Enable(FALSE);
    _eState                         := E_PROGRESS.PROGRESS_OCCUPIED;
END_CASE
CASE _eState
OF
  E_PROGRESS.PROGRESS_OCCUPIED:
    _eResult                        := Enable(TRUE);

    IF (_eResult = E_PROGRESS.PROGRESS_DONE)
    THEN
      _eState                       := E_PROGRESS.PROGRESS_WORKING;
    END_IF
END_CASE
CASE _eState
OF
  E_PROGRESS.PROGRESS_WORKING:
    _eState                         := E_PROGRESS.PROGRESS_DONE;
END_CASE

AxisEnable := _eState;
END_METHOD

METHOD AxisGearIn : E_PROGRESS
VAR_INPUT
  Execute           : BOOL;
END_VAR
VAR_INST
  _eState           : E_PROGRESS;
  _rValue           : LREAL;
  _nErr,
  _nMasterIndex,
  _nMasterNcId      : UDINT;
  _stMsg            : ST_Message;


END_VAR
IF NOT Check() THEN AxisGearIn := E_PROGRESS.PROGRESS_ERROR; RETURN; END_IF
IF NOT Execute THEN _eState := E_PROGRESS.PROGRESS_INIT; END_IF

CASE _eState
OF
  E_PROGRESS.PROGRESS_INIT:
    IF Execute 
    THEN
      memset(ADR(_stMsg),0,SIZEOF(_stMsg));
      _nMasterNcId                  :=
      _nMasterIndex                 :=
      _nErr                         := 0;
      _rValue                       := 0;

      IF NOT (_GearInParameter^[_nAxisIndex].nAxisIndexMaster[1] > 0) OR
         NOT (_GearInParameter^[_nAxisIndex].nAxisIndexMaster[1] < MAX_AXIS+1)
      THEN
        _nMasterIndex               := _GearInParameter^[_nAxisIndex].nAxisIndexMaster[1];

        _stMsg.eType                := E_MessageType.eMessageError;
        _stMsg.eDevice              := e_Device.Axis + TO_UINT(_AxisRef.NcToPlc.AxisId);
        _stMsg.eSubdevice           := e_Subdevice.fbGearIn;
        _stMsg.iErrorNumber         := 
        _nErr                       := 666;

        _stMsg.sText                := concat('_GearInParameter[', TO_STRING(_nAxisIndex));
        _stMsg.sText                := concat(_stMsg.sText,    '].nAxisIndexMaster[1] out of range: ');
        _stMsg.sText                := concat(_stMsg.sText, TO_STRING(_nMasterIndex));

        f_MessageSet(_stMsg);

        _eState                     := E_PROGRESS.PROGRESS_ERROR;

      ELSE
        _eState                     := E_PROGRESS.PROGRESS_BUSY;

        _nMasterIndex               := _GearInParameter^[_nAxisIndex].nAxisIndexMaster[1];
        _nMasterNcId                := _Info^[_nMasterIndex].nNcAxisId;

        _stMsg.eType                := E_MessageType.eMessageInfo;
        _stMsg.eDevice              := e_Device.Axis + TO_UINT(_AxisRef.NcToPlc.AxisId);
        _stMsg.eSubdevice           := e_Subdevice.fbGearIn;
        _stMsg.iErrorNumber         := 0;
  
        _stMsg.sText                := concat('GearIn BUSY: ', TO_STRING(_nMasterIndex));
        f_MessageSet(_stMsg);
      END_IF
    END_IF
END_CASE
CASE _eState
OF
  E_PROGRESS.PROGRESS_BUSY:
    _eState                         := E_PROGRESS.PROGRESS_STARTUP;
    _fbGearIn(
              Master                := _Axes[_nMasterIndex], 
              Slave                 := _AxisRef, 
              Execute               := FALSE, 
              RatioNumerator        := _GearInParameter^[_nAxisIndex].rGearRatio[1], 
              RatioDenominator      := 1, 
              Acceleration          := _GearInParameter^[_nAxisIndex].Acceleration, 
              Deceleration          := _GearInParameter^[_nAxisIndex].Deceleration, 
              Jerk                  := _GearInParameter^[_nAxisIndex].Jerk);
END_CASE
CASE _eState
OF
  E_PROGRESS.PROGRESS_STARTUP:
    _fbGearIn(
              Master                := _Axes[_nMasterIndex], 
              Slave                 := _AxisRef, 
              Execute               := TRUE, 
              RatioNumerator        := _GearInParameter^[_nAxisIndex].rGearRatio[1], 
              RatioDenominator      := 1, 
              Acceleration          := _GearInParameter^[_nAxisIndex].Acceleration, 
              Deceleration          := _GearInParameter^[_nAxisIndex].Deceleration, 
              Jerk                  := _GearInParameter^[_nAxisIndex].Jerk);

    IF (_fbGearIn.Error)
    THEN
      _nErr                         := _fbGearIn.ErrorID;

      _stMsg.eType                  := E_MessageType.eMessageError;
      _stMsg.eDevice                := e_Device.Axis + TO_UINT(_AxisRef.NcToPlc.AxisId);
      _stMsg.eSubdevice             := e_Subdevice.fbGearIn;
      _stMsg.iErrorNumber           := _nErr;

      _stMsg.sText                  := concat('GearIn ERROR: ', TO_STRING(_nMasterIndex));
      f_MessageSet(_stMsg);
      _eState                       := E_PROGRESS.PROGRESS_ERROR;

    ELSIF (_fbGearIn.InGear)
    THEN
      _eState                       := E_PROGRESS.PROGRESS_CHECK;
    END_IF
END_CASE
CASE _eState
OF
  E_PROGRESS.PROGRESS_CHECK:
    _eState                         := E_PROGRESS.PROGRESS_DONE;

    _stMsg.eType                    := E_MessageType.eMessageInfo;
    _stMsg.eDevice                  := e_Device.Axis + TO_UINT(_AxisRef.NcToPlc.AxisId);
    _stMsg.eSubdevice               := e_Subdevice.fbGearIn;
    _stMsg.iErrorNumber             := 0;

    _stMsg.sText                    := concat('GearIn done: ', TO_STRING(_nMasterIndex));
    f_MessageSet(_stMsg);
END_CASE
CASE _eState
OF
  E_PROGRESS.PROGRESS_DONE,
  E_PROGRESS.PROGRESS_ERROR:
    _fbGearIn(
              Master                := _Axes[_nMasterIndex], 
              Slave                 := _AxisRef, 
              Execute               := FALSE);
END_CASE

AxisGearIn                          := _eState;
END_METHOD

METHOD AxisGearInMultiMaster : E_PROGRESS
VAR_INPUT
  Execute           : BOOL;
END_VAR
VAR_INST
  _eState           : E_PROGRESS;
  _rValue           : LREAL;
  _nAx,
  _nErr             : UDINT;

  _nMasterIndex,
  _nMasterNcId      : ARRAY[1..4] OF UDINT;

  _stOptions        : Tc2_MC2.ST_GearInMultiMasterOptions;
  _nSyncMode        : int;

  _stMsg            : ST_Message;


END_VAR
IF NOT Check() THEN AxisGearInMultiMaster := E_PROGRESS.PROGRESS_ERROR; RETURN; END_IF
IF NOT Execute THEN _eState := E_PROGRESS.PROGRESS_INIT; END_IF

CASE _eState
OF
  E_PROGRESS.PROGRESS_INIT:
    IF Execute 
    THEN
      memset(ADR(_stMsg),0,SIZEOF(_stMsg));
      memset(ADR(_nMasterNcId), 0,SIZEOF(_nMasterNcId));
      memset(ADR(_nMasterIndex),0,SIZEOF(_nMasterIndex));
      memset(ADR(_stOptions),   0,SIZEOF(_stOptions));
      _nErr                           := 0;
      _rValue                         := 0;

      IF NOT (_GearInParameter^[_nAxisIndex].nAxisIndexMaster[1] > 0) OR
         NOT (_GearInParameter^[_nAxisIndex].nAxisIndexMaster[1] <= MAX_AXIS)
      THEN
        _nMasterIndex[1]              := _GearInParameter^[_nAxisIndex].nAxisIndexMaster[1];

        _stMsg.eType                  := E_MessageType.eMessageError;
        _stMsg.eDevice                := e_Device.Axis + TO_UINT(_AxisRef.NcToPlc.AxisId);
        _stMsg.eSubdevice             := e_Subdevice.fbGearInMultiMaster;
        _stMsg.iErrorNumber           := 
        _nErr                         := 666;

        _stMsg.sText                  := concat('_GearInParameter[', TO_STRING(_nAxisIndex));
        _stMsg.sText                  := concat(_stMsg.sText,    '].nAxisIndexMaster[1] out of range: ');
        _stMsg.sText                  := concat(_stMsg.sText, TO_STRING(_nMasterIndex[1]));
        f_MessageSet(_stMsg);

        _eState                       := E_PROGRESS.PROGRESS_ERROR;

      ELSE
        _eState                       := E_PROGRESS.PROGRESS_BUSY;

        _stOptions.AdvancedSlaveDynamics  := _GearInParameter^[_nAxisIndex].bAdvancedSlaveDynamics;
        _nSyncMode                        := _GearInParameter^[_nAxisIndex].nMultiMasterSyncMode;

        _nMasterIndex[1]              := _GearInParameter^[_nAxisIndex].nAxisIndexMaster[1];
        _nMasterNcId[1]               := _Info^[_nMasterIndex[1]].nNcAxisId;
        memcpy(ADR(_stOptions.SyncMode), ADR(_nSyncMode), SIZEOF(_stOptions.SyncMode));

        _fbGearInMultiMaster.Master1  := _Axes[_nMasterIndex[1]];   // assign AXIS_REF of master

        _stMsg.eType                  := E_MessageType.eMessageInfo;
        _stMsg.eDevice                := e_Device.Axis + TO_UINT(_AxisRef.NcToPlc.AxisId);
        _stMsg.eSubdevice             := e_Subdevice.fbGearInMultiMaster;
        _stMsg.iErrorNumber           := _eState;

        _stMsg.sText                  := concat('_GearInParameter[', TO_STRING(_nAxisIndex));
        _stMsg.sText                  := concat(_stMsg.sText,    '] MultiMaster check: ');
        _stMsg.sText                  := concat(_stMsg.sText, TO_STRING(_nMasterIndex[1]));
        f_MessageSet(_stMsg);

        _nAx                          := 2; // next master index to check
      END_IF
    END_IF
END_CASE
CASE _eState
OF
  E_PROGRESS.PROGRESS_BUSY:
    IF NOT (_GearInParameter^[_nAxisIndex].nAxisIndexMaster[_nAx] > 0) OR
       NOT (_GearInParameter^[_nAxisIndex].nAxisIndexMaster[_nAx] < MAX_AXIS+1)
    THEN
      // next entry not valid
      // Master1 is already checked --> let's get ready
      _eState                         := E_PROGRESS.PROGRESS_CHECK;
    ELSE
      _eState                         := E_PROGRESS.PROGRESS_STARTUP;

      _nMasterIndex[_nAx]             := _GearInParameter^[_nAxisIndex].nAxisIndexMaster[_nAx];
      _nMasterNcId [_nAx]             := _Info^[_nMasterIndex[_nAx]].nNcAxisId;

      _stMsg.eType                    := E_MessageType.eMessageInfo;
      _stMsg.eDevice                  := e_Device.Axis + TO_UINT(_AxisRef.NcToPlc.AxisId);
      _stMsg.eSubdevice               := e_Subdevice.fbGearInMultiMaster;
      _stMsg.iErrorNumber             := _eState;

      _stMsg.sText                    := concat('_GearInParameter[', TO_STRING(_nAxisIndex));
      _stMsg.sText                    := concat(_stMsg.sText,    '] MultiMaster check: ');
      _stMsg.sText                    := concat(_stMsg.sText, TO_STRING(_nMasterIndex[_nAx]));
      f_MessageSet(_stMsg);
    END_IF

    _fbGearInMultiMaster(
                      Slave           := _AxisRef, 
                      Enable          := FALSE, 
                      GearRatio1      := _GearInParameter^[_nAxisIndex].rGearRatio[1], 
                      GearRatio2      := _GearInParameter^[_nAxisIndex].rGearRatio[2], 
                      GearRatio3      := _GearInParameter^[_nAxisIndex].rGearRatio[3], 
                      GearRatio4      := _GearInParameter^[_nAxisIndex].rGearRatio[4], 
                      Acceleration    := _GearInParameter^[_nAxisIndex].Acceleration, 
                      Deceleration    := _GearInParameter^[_nAxisIndex].Deceleration, 
                      Jerk            := _GearInParameter^[_nAxisIndex].Jerk,
                      Options         := _stOptions);
END_CASE
CASE _eState
OF
  E_PROGRESS.PROGRESS_STARTUP:
    CASE _nAx
    OF
      2:
        _nAx                          := _nAx + 1;
        _eState                       := E_PROGRESS.PROGRESS_BUSY;
        _fbGearInMultiMaster.Master2  := _Axes[_nMasterIndex[2]];   // assign AXIS_REF of master

      3:
        _nAx                          := _nAx + 1;
        _eState                       := E_PROGRESS.PROGRESS_BUSY;
        _fbGearInMultiMaster.Master3  := _Axes[_nMasterIndex[3]];   // assign AXIS_REF of master

